C03625=1090.192,-119.581,450.543,174.558,16.064,152.527
C03626=1090.198,-119.332,450.534,174.560,16.065,152.526
C03627=1090.205,-119.082,450.524,174.562,16.066,152.526
C03628=1090.211,-118.832,450.515,174.563,16.066,152.526
C03629=1090.217,-118.582,450.505,174.565,16.066,152.526
C03630=1090.223,-118.332,450.496,174.567,16.067,152.525
C03631=1090.229,-118.082,450.487,174.568,16.067,152.525
C03632=1090.235,-117.832,450.477,174.570,16.068,152.525
C03633=1090.241,-117.583,450.468,174.571,16.069,152.525
C03634=1090.247,-117.333,450.458,174.573,16.069,152.525
C03635=1090.253,-117.084,450.449,174.574,16.070,152.524
C03636=1090.259,-116.834,450.439,174.576,16.070,152.524
C03637=1090.265,-116.584,450.430,174.577,16.070,152.524
C03638=1090.272,-116.334,450.420,174.579,16.071,152.524
C03639=1090.279,-116.085,450.411,174.580,16.071,152.523
C03640=1090.285,-115.835,450.402,174.582,16.072,152.523
C03641=1090.291,-115.585,450.392,174.584,16.073,152.523
C03642=1090.297,-115.335,450.382,174.585,16.073,152.523
C03643=1090.303,-115.086,450.373,174.587,16.073,152.522
C03644=1090.309,-114.836,450.364,174.589,16.074,152.522
C03645=1090.315,-114.587,450.354,174.590,16.074,152.522
C03646=1090.321,-114.337,450.345,174.592,16.075,152.522
C03647=1090.327,-114.087,450.335,174.594,16.076,152.522
C03648=1090.333,-113.837,450.325,174.595,16.076,152.521
C03649=1090.340,-113.587,450.316,174.597,16.076,152.521
C03650=1090.345,-113.318,450.306,174.598,16.077,152.521
C03651=1090.352,-113.049,450.295,174.600,16.078,152.521
C03652=1090.359,-112.781,450.285,174.601,16.078,152.521
C03653=1090.365,-112.512,450.275,174.603,16.079,152.520
C03654=1090.371,-112.262,450.265,174.605,16.080,152.520
C03655=1090.378,-112.012,450.256,174.607,16.080,152.520
C03656=1090.384,-111.762,450.246,174.608,16.080,152.519
C03657=1090.390,-111.513,450.236,174.610,16.081,152.519
C03658=1090.396,-111.263,450.226,174.612,16.082,152.519
C03659=1090.402,-111.013,450.216,174.613,16.082,152.519
C03660=1090.408,-110.763,450.207,174.615,16.083,152.519
C03661=1090.414,-110.514,450.197,174.616,16.084,152.519
C03662=1090.420,-110.264,450.188,174.617,16.084,152.518
C03663=1090.427,-110.014,450.178,174.619,16.085,152.518
C03664=1090.433,-109.764,450.168,174.621,16.085,152.518
C03665=1090.439,-109.514,450.159,174.622,16.086,152.518
C03666=1090.445,-109.265,450.149,174.624,16.086,152.517
C03667=1090.451,-109.015,450.140,174.626,16.087,152.517
C03668=1090.458,-108.766,450.130,174.627,16.087,152.517
C03669=1090.464,-108.516,450.120,174.628,16.088,152.517
C03670=1090.470,-108.266,450.110,174.630,16.089,152.517
C03671=1090.475,-108.016,450.100,174.632,16.089,152.516
C03672=1090.482,-107.766,450.091,174.633,16.089,152.516
C03673=1090.488,-107.516,450.081,174.635,16.091,152.516
C03674=1090.494,-107.266,450.072,174.637,16.091,152.516
C03675=1090.500,-107.017,450.061,174.638,16.091,152.515
C03676=1090.507,-106.767,450.052,174.640,16.092,152.515
C03677=1090.512,-106.517,450.041,174.641,16.093,152.515
C03678=1090.518,-106.268,450.032,174.643,16.093,152.515
C03679=1090.524,-106.018,450.023,174.644,16.094,152.515
C03680=1090.530,-105.769,450.013,174.646,16.095,152.515
C03681=1090.536,-105.519,450.003,174.648,16.096,152.514
C03682=1090.542,-105.269,449.993,174.649,16.096,152.514
C03683=1090.548,-105.020,449.983,174.651,16.097,152.514
C03684=1090.554,-104.770,449.974,174.653,16.097,152.514
C03685=1090.561,-104.521,449.963,174.653,16.098,152.514
C03686=1090.566,-104.271,449.953,174.655,16.099,152.513
C03687=1090.572,-104.021,449.944,174.657,16.099,152.513
C03688=1090.579,-103.771,449.934,174.659,16.100,152.513
C03689=1090.585,-103.521,449.924,174.660,16.100,152.513
C03690=1090.591,-103.272,449.914,174.662,16.101,152.512
C03691=1090.597,-103.022,449.904,174.663,16.102,152.512
C03692=1090.603,-102.772,449.894,174.665,16.103,152.512
C03693=1090.609,-102.522,449.885,174.666,16.103,152.512
C03694=1090.615,-102.273,449.874,174.668,16.104,152.512
C03695=1090.621,-102.023,449.864,174.670,16.105,152.511
C03696=1090.627,-101.773,449.855,174.672,16.106,152.511
C03697=1090.634,-101.523,449.844,174.673,16.106,152.511
C03698=1090.640,-101.273,449.834,174.675,16.106,152.511
C03699=1090.646,-101.023,449.824,174.676,16.108,152.511
C03700=1090.652,-100.774,449.814,174.677,16.108,152.511
C03701=1090.658,-100.524,449.805,174.679,16.108,152.510
C03702=1090.664,-100.274,449.794,174.681,16.109,152.510
C03703=1090.670,-100.024,449.785,174.683,16.110,152.510
C03704=1090.676,-99.775,449.775,174.684,16.111,152.510
C03705=1090.682,-99.525,449.764,174.685,16.111,152.510
C03706=1090.688,-99.276,449.754,174.687,16.112,152.509
C03707=1090.695,-99.026,449.745,174.689,16.113,152.509
C03708=1090.700,-98.776,449.734,174.690,16.113,152.509
C03709=1090.706,-98.527,449.724,174.692,16.114,152.509
C03710=1090.713,-98.277,449.715,174.694,16.115,152.509
C03711=1090.719,-98.027,449.705,174.696,16.115,152.508
C03712=1090.725,-97.778,449.694,174.696,16.116,152.508
C03713=1090.731,-97.528,449.685,174.698,16.117,152.508
C03714=1090.738,-97.252,449.673,174.700,16.118,152.508
C03715=1090.744,-96.976,449.662,174.702,16.118,152.508
C03716=1090.750,-96.701,449.651,174.703,16.120,152.508
C03717=1090.756,-96.425,449.640,174.705,16.120,152.507
C03718=1090.764,-96.175,449.629,174.707,16.121,152.507
C03719=1090.770,-95.925,449.619,174.709,16.122,152.507
C03720=1090.775,-95.676,449.608,174.710,16.123,152.507
C03721=1090.782,-95.426,449.599,174.712,16.123,152.507
C03722=1090.787,-95.176,449.589,174.713,16.124,152.506
C03723=1090.793,-94.927,449.578,174.715,16.125,152.506
C03724=1090.799,-94.677,449.568,174.716,16.126,152.506
C03725=1090.805,-94.427,449.558,174.718,16.126,152.506
C03726=1090.811,-94.177,449.548,174.719,16.127,152.506
C03727=1090.817,-93.928,449.538,174.721,16.128,152.505
C03728=1090.823,-93.678,449.527,174.723,16.129,152.505
C03729=1090.829,-93.429,449.517,174.724,16.129,152.505
C03730=1090.835,-93.179,449.507,174.726,16.130,152.505
C03731=1090.841,-92.930,449.497,174.727,16.131,152.505
C03732=1090.847,-92.680,449.487,174.729,16.132,152.505
C03733=1090.854,-92.430,449.476,174.731,16.133,152.504
C03734=1090.859,-92.180,449.466,174.732,16.133,152.504
C03735=1090.865,-91.930,449.455,174.734,16.134,152.504
C03736=1090.871,-91.680,449.445,174.735,16.135,152.504
C03737=1090.877,-91.431,449.434,174.737,16.136,152.504
C03738=1090.883,-91.181,449.425,174.739,16.137,152.504
C03739=1090.889,-90.931,449.414,174.740,16.137,152.504
C03740=1090.895,-90.682,449.404,174.742,16.138,152.503
C03741=1090.901,-90.432,449.394,174.743,16.139,152.503
C03742=1090.907,-90.182,449.384,174.745,16.140,152.503
C03743=1090.913,-89.932,449.373,174.747,16.141,152.503
C03744=1090.920,-89.683,449.362,174.748,16.141,152.503
C03745=1090.925,-89.433,449.352,174.749,16.142,152.502
C03746=1090.931,-89.184,449.342,174.751,16.143,152.502
C03747=1090.937,-88.934,449.332,174.753,16.144,152.502
C03748=1090.943,-88.684,449.321,174.755,16.145,152.502
C03749=1090.950,-88.434,449.310,174.756,16.145,152.502
C03750=1090.955,-88.184,449.300,174.757,16.146,152.502
C03751=1090.962,-87.935,449.290,174.759,16.147,152.501
C03752=1090.967,-87.685,449.280,174.761,16.148,152.501
C03753=1090.974,-87.436,449.269,174.762,16.149,152.501
C03754=1090.979,-87.186,449.259,174.763,16.149,152.501
C03755=1090.985,-86.935,449.248,174.765,16.150,152.501
C03756=1090.992,-86.686,449.238,174.767,16.151,152.501
C03757=1090.998,-86.437,449.227,174.769,16.152,152.500
C03758=1091.004,-86.187,449.217,174.771,16.153,152.500
C03759=1091.009,-85.937,449.206,174.772,16.154,152.500
C03760=1091.016,-85.687,449.195,174.773,16.154,152.500
C03761=1091.022,-85.437,449.186,174.775,16.155,152.500
C03762=1091.028,-85.188,449.175,174.776,16.156,152.500
C03763=1091.034,-84.939,449.164,174.778,16.157,152.499
C03764=1091.040,-84.689,449.154,174.780,16.158,152.499
C03765=1091.046,-84.438,449.143,174.782,16.159,152.499
C03766=1091.052,-84.189,449.133,174.783,16.159,152.499
C03767=1091.058,-83.940,449.122,174.784,16.160,152.499
C03768=1091.064,-83.690,449.112,174.786,16.161,152.499
C03769=1091.070,-83.440,449.101,174.788,16.162,152.498
C03770=1091.076,-83.190,449.090,174.789,16.163,152.498
C03771=1091.083,-82.941,449.080,174.791,16.164,152.498
C03772=1091.088,-82.691,449.070,174.792,16.164,152.498
C03773=1091.094,-82.442,449.059,174.794,16.165,152.498
C03774=1091.101,-82.192,449.048,174.796,16.166,152.498
C03775=1091.107,-81.942,449.037,174.797,16.167,152.498
C03776=1091.113,-81.692,449.028,174.799,16.168,152.497
C03777=1091.119,-81.443,449.017,174.801,16.169,152.497
C03778=1091.126,-81.170,449.005,174.803,16.170,152.497
C03779=1091.132,-80.896,448.993,174.804,16.171,152.497
C03780=1091.139,-80.623,448.981,174.806,16.172,152.497
C03781=1091.146,-80.349,448.970,174.808,16.173,152.496
C03782=1091.152,-80.099,448.960,174.809,16.174,152.496
C03783=1091.157,-79.850,448.949,174.811,16.175,152.496
C03784=1091.164,-79.600,448.937,174.812,16.175,152.496
C03785=1091.170,-79.350,448.927,174.814,16.176,152.496
C03786=1091.176,-79.101,448.916,174.815,16.177,152.496
C03787=1091.181,-78.851,448.906,174.817,16.178,152.496
C03788=1091.188,-78.601,448.895,174.819,16.179,152.495
C03789=1091.193,-78.351,448.884,174.820,16.180,152.495
C03790=1091.200,-78.102,448.874,174.822,16.181,152.495
C03791=1091.206,-77.852,448.863,174.823,16.181,152.495
C03792=1091.212,-77.602,448.852,174.825,16.183,152.495
C03793=1091.218,-77.353,448.841,174.826,16.184,152.495
C03794=1091.223,-77.103,448.831,174.828,16.184,152.495
C03795=1091.229,-76.853,448.820,174.830,16.185,152.494
C03796=1091.236,-76.603,448.809,174.832,16.187,152.494
C03797=1091.242,-76.354,448.798,174.833,16.187,152.494
C03798=1091.247,-76.104,448.787,174.835,16.188,152.494
C03799=1091.253,-75.855,448.776,174.837,16.190,152.494
C03800=1091.260,-75.605,448.765,174.837,16.190,152.494
C03801=1091.265,-75.355,448.754,174.839,16.191,152.494
C03802=1091.271,-75.106,448.743,174.841,16.192,152.493
C03803=1091.278,-74.856,448.733,174.843,16.193,152.493
C03804=1091.284,-74.606,448.722,174.844,16.194,152.493
C03805=1091.290,-74.357,448.711,174.846,16.195,152.493
C03806=1091.296,-74.107,448.700,174.848,16.196,152.493
C03807=1091.302,-73.857,448.689,174.849,16.197,152.493
C03808=1091.307,-73.608,448.678,174.851,16.198,152.493
C03809=1091.313,-73.358,448.668,174.852,16.198,152.492
C03810=1091.319,-73.108,448.657,174.854,16.199,152.492
C03811=1091.325,-72.858,448.646,174.855,16.201,152.492
C03812=1091.331,-72.608,448.635,174.857,16.202,152.492
C03813=1091.336,-72.359,448.624,174.859,16.203,152.492
C03814=1091.342,-72.109,448.613,174.860,16.204,152.492
C03815=1091.348,-71.859,448.602,174.862,16.205,152.492
C03816=1091.354,-71.610,448.591,174.864,16.206,152.491
C03817=1091.360,-71.360,448.580,174.865,16.207,152.491
C03818=1091.366,-71.110,448.568,174.867,16.208,152.491
C03819=1091.372,-70.861,448.557,174.868,16.209,152.491
C03820=1091.377,-70.611,448.546,174.869,16.210,152.491
C03821=1091.383,-70.362,448.535,174.871,16.210,152.491
C03822=1091.389,-70.112,448.524,174.873,16.212,152.491
C03823=1091.395,-69.862,448.513,174.874,16.213,152.491
C03824=1091.401,-69.613,448.502,174.876,16.214,152.491
C03825=1091.407,-69.362,448.491,174.878,16.215,152.490
C03826=1091.413,-69.113,448.480,174.879,16.216,152.490
C03827=1091.419,-68.863,448.469,174.881,16.217,152.490
C03828=1091.425,-68.613,448.458,174.883,16.218,152.490
C03829=1091.431,-68.364,448.447,174.884,16.219,152.490
C03830=1091.437,-68.114,448.436,174.886,16.220,152.490
C03831=1091.442,-67.864,448.424,174.888,16.221,152.490
C03832=1091.448,-67.615,448.413,174.889,16.222,152.490
C03833=1091.454,-67.365,448.402,174.891,16.224,152.489
C03834=1091.460,-67.115,448.390,174.892,16.224,152.489
C03835=1091.466,-66.866,448.380,174.894,16.225,152.489
C03836=1091.472,-66.616,448.369,174.895,16.226,152.489
C03837=1091.478,-66.366,448.357,174.897,16.227,152.489
C03838=1091.484,-66.117,448.347,174.898,16.228,152.489
C03839=1091.490,-65.868,448.335,174.900,16.229,152.489
C03840=1091.495,-65.617,448.323,174.902,16.230,152.488
C03841=1091.501,-65.368,448.312,174.903,16.231,152.488
C03842=1091.508,-65.097,448.300,174.905,16.232,152.488
C03843=1091.514,-64.825,448.288,174.907,16.233,152.488
C03844=1091.521,-64.555,448.276,174.908,16.235,152.488
C03845=1091.528,-64.283,448.264,174.911,16.236,152.488
C03846=1091.533,-64.033,448.253,174.912,16.237,152.488
C03847=1091.539,-63.784,448.241,174.913,16.237,152.488
C03848=1091.545,-63.534,448.229,174.915,16.239,152.487
C03849=1091.551,-63.284,448.218,174.917,16.240,152.487
C03850=1091.557,-63.034,448.207,174.918,16.241,152.487
C03851=1091.563,-62.785,448.196,174.920,16.242,152.487
C03852=1091.569,-62.536,448.185,174.921,16.243,152.487
C03853=1091.575,-62.286,448.173,174.923,16.244,152.487
C03854=1091.580,-62.036,448.162,174.925,16.245,152.487
C03855=1091.587,-61.786,448.150,174.927,16.246,152.487
C03856=1091.593,-61.537,448.139,174.928,16.247,152.486
C03857=1091.598,-61.287,448.128,174.930,16.248,152.486
C03858=1091.605,-61.037,448.117,174.931,16.249,152.486
C03859=1091.610,-60.788,448.105,174.933,16.251,152.486
C03860=1091.616,-60.538,448.094,174.935,16.252,152.486
C03861=1091.622,-60.288,448.083,174.936,16.253,152.486
C03862=1091.629,-60.039,448.071,174.938,16.254,152.486
C03863=1091.634,-59.789,448.060,174.940,16.255,152.486
C03864=1091.641,-59.539,448.049,174.941,16.256,152.485
C03865=1091.646,-59.290,448.036,174.943,16.257,152.485
C03866=1091.652,-59.039,448.025,174.945,16.258,152.485
C03867=1091.658,-58.790,448.014,174.946,16.259,152.485
C03868=1091.665,-58.540,448.002,174.948,16.260,152.485
C03869=1091.670,-58.291,447.991,174.949,16.262,152.485
C03870=1091.677,-58.041,447.979,174.951,16.262,152.485
C03871=1091.682,-57.792,447.968,174.953,16.263,152.485
C03872=1091.688,-57.542,447.957,174.955,16.264,152.484
C03873=1091.695,-57.293,447.945,174.956,16.266,152.484
C03874=1091.700,-57.042,447.933,174.958,16.267,152.484
C03875=1091.706,-56.793,447.922,174.959,16.268,152.484
C03876=1091.713,-56.543,447.911,174.961,16.269,152.484
C03877=1091.718,-56.293,447.900,174.963,16.270,152.484
C03878=1091.724,-56.044,447.887,174.964,16.271,152.484
C03879=1091.730,-55.794,447.876,174.966,16.272,152.484
C03880=1091.737,-55.544,447.864,174.968,16.273,152.483
C03881=1091.742,-55.295,447.853,174.969,16.274,152.483
C03882=1091.748,-55.045,447.841,174.971,16.275,152.483
C03883=1091.754,-54.796,447.830,174.973,16.276,152.483
C03884=1091.761,-54.546,447.818,174.974,16.278,152.483
C03885=1091.766,-54.297,447.807,174.976,16.279,152.483
C03886=1091.772,-54.047,447.795,174.977,16.280,152.483
C03887=1091.778,-53.797,447.784,174.979,16.281,152.483
C03888=1091.785,-53.548,447.772,174.981,16.282,152.482
C03889=1091.791,-53.297,447.761,174.983,16.283,152.482
C03890=1091.796,-53.048,447.748,174.984,16.284,152.482
C03891=1091.803,-52.798,447.737,174.986,16.285,152.482
C03892=1091.809,-52.549,447.725,174.987,16.286,152.482
C03893=1091.814,-52.299,447.714,174.989,16.287,152.482
C03894=1091.820,-52.050,447.702,174.991,16.289,152.482
C03895=1091.827,-51.800,447.691,174.992,16.290,152.482
C03896=1091.833,-51.550,447.679,174.994,16.290,152.481
C03897=1091.839,-51.301,447.667,174.996,16.291,152.481
C03898=1091.845,-51.051,447.655,174.997,16.293,152.481
C03899=1091.851,-50.802,447.644,174.999,16.294,152.481
C03900=1091.857,-50.551,447.632,175.001,16.295,152.481
C03901=1091.863,-50.302,447.620,175.002,16.296,152.481
C03902=1091.868,-50.052,447.609,175.004,16.297,152.481
C03903=1091.875,-49.802,447.597,175.005,16.298,152.481
C03904=1091.880,-49.553,447.584,175.007,16.299,152.481
C03905=1091.887,-49.303,447.573,175.009,16.301,152.480
C03906=1091.893,-49.034,447.560,175.010,16.302,152.480
C03907=1091.899,-48.763,447.547,175.012,16.303,152.480
C03908=1091.905,-48.493,447.535,175.013,16.304,152.480
C03909=1091.911,-48.224,447.522,175.016,16.306,152.480
C03910=1091.918,-47.974,447.510,175.017,16.307,152.480
C03911=1091.923,-47.724,447.498,175.019,16.308,152.480
C03912=1091.930,-47.475,447.486,175.021,16.309,152.480
C03913=1091.935,-47.225,447.474,175.022,16.310,152.480
C03914=1091.941,-46.975,447.462,175.024,16.311,152.480
C03915=1091.947,-46.726,447.451,175.026,16.313,152.479
C03916=1091.953,-46.476,447.438,175.027,16.314,152.479
C03917=1091.959,-46.227,447.426,175.029,16.315,152.479
C03918=1091.964,-45.977,447.415,175.030,16.316,152.479
C03919=1091.971,-45.727,447.403,175.032,16.317,152.479
C03920=1091.976,-45.478,447.391,175.034,16.318,152.479
C03921=1091.982,-45.228,447.379,175.035,16.319,152.479
C03922=1091.988,-44.978,447.367,175.037,16.320,152.479
C03923=1091.994,-44.729,447.355,175.038,16.322,152.479
C03924=1092.000,-44.479,447.343,175.040,16.323,152.478
C03925=1092.005,-44.229,447.331,175.042,16.324,152.478
C03926=1092.011,-43.979,447.319,175.043,16.325,152.478
C03927=1092.018,-43.730,447.307,175.045,16.326,152.478
C03928=1092.023,-43.481,447.295,175.046,16.327,152.478
C03929=1092.030,-43.231,447.283,175.048,16.328,152.478
C03930=1092.036,-42.981,447.271,175.050,16.330,152.478
C03931=1092.041,-42.731,447.259,175.052,16.331,152.478
C03932=1092.047,-42.482,447.247,175.054,16.332,152.478
C03933=1092.053,-42.231,447.235,175.055,16.334,152.477
C03934=1092.059,-41.983,447.223,175.057,16.335,152.477
C03935=1092.065,-41.733,447.211,175.059,16.336,152.477
C03936=1092.070,-41.483,447.198,175.060,16.337,152.477
C03937=1092.077,-41.234,447.187,175.062,16.338,152.477
C03938=1092.083,-40.984,447.174,175.063,16.339,152.477
C03939=1092.088,-40.734,447.162,175.065,16.340,152.477
C03940=1092.095,-40.485,447.151,175.067,16.342,152.477
C03941=1092.100,-40.235,447.138,175.068,16.343,152.477
C03942=1092.107,-39.985,447.126,175.070,16.344,152.477
C03943=1092.112,-39.736,447.114,175.071,16.345,152.476
C03944=1092.118,-39.486,447.101,175.073,16.346,152.476
C03945=1092.125,-39.237,447.089,175.075,16.347,152.476
C03946=1092.130,-38.987,447.077,175.077,16.349,152.476
C03947=1092.136,-38.737,447.065,175.079,16.350,152.476
C03948=1092.143,-38.487,447.053,175.080,16.351,152.476
C03949=1092.148,-38.238,447.041,175.082,16.352,152.476
C03950=1092.154,-37.988,447.029,175.084,16.354,152.476
C03951=1092.160,-37.738,447.016,175.085,16.355,152.476
C03952=1092.165,-37.489,447.004,175.087,16.356,152.476
C03953=1092.171,-37.239,446.991,175.088,16.357,152.475
C03954=1092.178,-36.990,446.979,175.090,16.358,152.475
C03955=1092.183,-36.741,446.967,175.092,16.359,152.475
C03956=1092.189,-36.491,446.955,175.093,16.360,152.475
C03957=1092.195,-36.241,446.942,175.095,16.362,152.475
C03958=1092.200,-35.992,446.930,175.097,16.364,152.475
C03959=1092.207,-35.742,446.918,175.099,16.365,152.475
C03960=1092.212,-35.492,446.905,175.100,16.366,152.475
C03961=1092.218,-35.243,446.893,175.102,16.367,152.475
C03962=1092.224,-34.993,446.881,175.103,16.368,152.475
C03963=1092.230,-34.743,446.868,175.105,16.369,152.474
C03964=1092.236,-34.493,446.855,175.107,16.371,152.474
C03965=1092.242,-34.244,446.844,175.108,16.372,152.474
C03966=1092.247,-33.995,446.831,175.110,16.373,152.474
C03967=1092.253,-33.745,446.819,175.111,16.374,152.474
C03968=1092.259,-33.495,446.807,175.114,16.376,152.474
C03969=1092.265,-33.246,446.794,175.115,16.377,152.474
C03970=1092.271,-32.976,446.781,175.117,16.378,152.474
C03971=1092.277,-32.707,446.767,175.119,16.379,152.474
C03972=1092.284,-32.437,446.754,175.120,16.380,152.474
C03973=1092.290,-32.167,446.740,175.123,16.382,152.473
C03974=1092.296,-31.918,446.728,175.124,16.383,152.473
C03975=1092.302,-31.668,446.715,175.126,16.385,152.473
C03976=1092.308,-31.418,446.703,175.127,16.386,152.473
C03977=1092.314,-31.168,446.690,175.129,16.387,152.473
C03978=1092.319,-30.919,446.678,175.130,16.388,152.473
C03979=1092.325,-30.669,446.666,175.132,16.389,152.473
C03980=1092.331,-30.420,446.653,175.135,16.391,152.473
C03981=1092.337,-30.170,446.641,175.136,16.392,152.473
C03982=1092.343,-29.920,446.627,175.138,16.393,152.473
C03983=1092.349,-29.671,446.615,175.139,16.394,152.472
C03984=1092.355,-29.422,446.603,175.141,16.396,152.472
C03985=1092.361,-29.172,446.591,175.143,16.397,152.472
C03986=1092.367,-28.922,446.578,175.144,16.398,152.472
C03987=1092.373,-28.672,446.565,175.146,16.399,152.472
C03988=1092.379,-28.423,446.553,175.147,16.400,152.472
C03989=1092.384,-28.174,446.540,175.150,16.402,152.472
C03990=1092.390,-27.924,446.527,175.151,16.403,152.472
C03991=1092.396,-27.674,446.515,175.153,16.404,152.472
C03992=1092.402,-27.424,446.502,175.155,16.405,152.472
C03993=1092.408,-27.175,446.489,175.156,16.406,152.471
C03994=1092.414,-26.925,446.477,175.158,16.408,152.471
C03995=1092.420,-26.676,446.464,175.160,16.409,152.471
C03996=1092.425,-26.426,446.452,175.161,16.410,152.471
C03997=1092.432,-26.176,446.439,175.163,16.412,152.471
C03998=1092.438,-25.927,446.426,175.165,16.413,152.471
C03999=1092.443,-25.677,446.414,175.166,16.414,152.471
C04000=1092.449,-25.427,446.401,175.168,16.416,152.471
C04001=1092.455,-25.178,446.388,175.170,16.417,152.471
C04002=1092.461,-24.928,446.375,175.171,16.418,152.471
C04003=1092.466,-24.678,446.362,175.173,16.419,152.471
C04004=1092.471,-24.429,446.350,175.175,16.421,152.470
C04005=1092.478,-24.180,446.337,175.177,16.422,152.470
C04006=1092.484,-23.930,446.324,175.179,16.423,152.470
C04007=1092.489,-23.680,446.312,175.180,16.424,152.470
C04008=1092.496,-23.431,446.298,175.181,16.426,152.470
C04009=1092.501,-23.181,446.286,175.183,16.427,152.470
C04010=1092.507,-22.932,446.274,175.185,16.428,152.470
C04011=1092.512,-22.682,446.260,175.187,16.430,152.470
C04012=1092.518,-22.432,446.247,175.189,16.431,152.470
C04013=1092.524,-22.182,446.235,175.190,16.432,152.470
C04014=1092.530,-21.933,446.221,175.192,16.433,152.469
C04015=1092.536,-21.683,446.209,175.194,16.434,152.469
C04016=1092.542,-21.435,446.196,175.195,16.435,152.469
C04017=1092.548,-21.185,446.183,175.198,16.437,152.469
C04018=1092.553,-20.934,446.170,175.199,16.438,152.469
C04019=1092.559,-20.685,446.157,175.201,16.439,152.469
C04020=1092.565,-20.435,446.144,175.202,16.441,152.469
C04021=1092.571,-20.186,446.131,175.204,16.442,152.469
C04022=1092.577,-19.936,446.119,175.205,16.443,152.469
C04023=1092.583,-19.686,446.106,175.208,16.445,152.469
C04024=1092.589,-19.437,446.092,175.209,16.446,152.469
C04025=1092.595,-19.187,446.080,175.211,16.447,152.468
C04026=1092.600,-18.938,446.067,175.213,16.448,152.468
C04027=1092.606,-18.688,446.054,175.214,16.450,152.468
C04028=1092.612,-18.439,446.041,175.216,16.451,152.468
C04029=1092.617,-18.189,446.028,175.217,16.452,152.468
C04030=1092.624,-17.940,446.014,175.220,16.454,152.468
C04031=1092.630,-17.690,446.002,175.221,16.455,152.468
C04032=1092.636,-17.440,445.989,175.223,16.456,152.468
C04033=1092.642,-17.191,445.976,175.225,16.457,152.468
C04034=1092.648,-16.921,445.962,175.227,16.459,152.467
C04035=1092.654,-16.650,445.947,175.229,16.460,152.467
C04036=1092.660,-16.379,445.934,175.230,16.461,152.467
C04037=1092.667,-16.109,445.919,175.233,16.463,152.467
C04038=1092.673,-15.859,445.906,175.234,16.464,152.467
C04039=1092.679,-15.610,445.893,175.236,16.465,152.467
C04040=1092.685,-15.361,445.880,175.237,16.467,152.467
C04041=1092.690,-15.110,445.867,175.239,16.468,152.467
C04042=1092.697,-14.861,445.853,175.241,16.469,152.467
C04043=1092.702,-14.612,445.841,175.243,16.471,152.467
C04044=1092.707,-14.362,445.827,175.245,16.472,152.466
C04045=1092.713,-14.112,445.815,175.246,16.473,152.466
C04046=1092.719,-13.863,445.801,175.248,16.474,152.466
C04047=1092.725,-13.614,445.788,175.249,16.475,152.466
C04048=1092.731,-13.364,445.775,175.252,16.477,152.466
C04049=1092.736,-13.114,445.761,175.253,16.478,152.466
C04050=1092.742,-12.864,445.749,175.255,16.479,152.466
C04051=1092.748,-12.615,445.735,175.256,16.481,152.466
C04052=1092.754,-12.365,445.721,175.258,16.482,152.466
C04053=1092.760,-12.115,445.709,175.260,16.484,152.466
C04054=1092.765,-11.866,445.695,175.262,16.485,152.466
C04055=1092.772,-11.617,445.682,175.264,16.486,152.465
C04056=1092.777,-11.366,445.669,175.265,16.487,152.465
C04057=1092.783,-11.117,445.655,175.267,16.488,152.465
C04058=1092.789,-10.868,445.642,175.269,16.490,152.465
C04059=1092.794,-10.618,445.629,175.271,16.491,152.465
C04060=1092.801,-10.368,445.616,175.272,16.492,152.465
C04061=1092.806,-10.119,445.602,175.274,16.493,152.465
C04062=1092.812,-9.870,445.589,175.276,16.494,152.465
C04063=1092.817,-9.619,445.575,175.278,16.496,152.465
C04064=1092.824,-9.370,445.562,175.279,16.498,152.465
C04065=1092.830,-9.121,445.549,175.281,16.499,152.465
C04066=1092.835,-8.871,445.536,175.283,16.500,152.464
C04067=1092.841,-8.621,445.522,175.284,16.501,152.464
C04068=1092.847,-8.372,445.509,175.287,16.503,152.464
C04069=1092.853,-8.123,445.495,175.288,16.504,152.464
C04070=1092.858,-7.873,445.481,175.290,16.505,152.464
C04071=1092.864,-7.623,445.469,175.292,16.506,152.464
C04072=1092.870,-7.374,445.455,175.293,16.508,152.464
C04073=1092.876,-7.124,445.442,175.296,16.509,152.464
C04074=1092.881,-6.875,445.428,175.297,16.510,152.464
C04075=1092.888,-6.625,445.415,175.299,16.512,152.463
C04076=1092.893,-6.375,445.401,175.300,16.513,152.463
C04077=1092.899,-6.126,445.388,175.302,16.514,152.463
C04078=1092.905,-5.876,445.374,175.304,16.516,152.463
C04079=1092.911,-5.626,445.361,175.306,16.517,152.463
C04080=1092.917,-5.377,445.347,175.308,16.518,152.463
C04081=1092.923,-5.128,445.334,175.309,16.519,152.463
C04082=1092.928,-4.877,445.320,175.312,16.521,152.463
C04083=1092.934,-4.628,445.307,175.313,16.522,152.463
C04084=1092.940,-4.379,445.293,175.315,16.523,152.462
C04085=1092.946,-4.129,445.280,175.317,16.524,152.462
C04086=1092.952,-3.880,445.266,175.318,16.525,152.462
C04087=1092.958,-3.631,445.253,175.321,16.527,152.462
C04088=1092.964,-3.380,445.239,175.322,16.528,152.462
C04089=1092.970,-3.131,445.225,175.324,16.529,152.462
C04090=1092.976,-2.881,445.212,175.325,16.530,152.462
C04091=1092.981,-2.632,445.198,175.328,16.533,152.462
C04092=1092.987,-2.382,445.184,175.329,16.534,152.462
C04093=1092.992,-2.132,445.171,175.331,16.535,152.462
C04094=1092.998,-1.883,445.157,175.332,16.536,152.462
C04095=1093.003,-1.633,445.143,175.335,16.538,152.461
C04096=1093.010,-1.384,445.130,175.336,16.539,152.461
C04097=1093.015,-1.134,445.116,175.338,16.540,152.461
C04098=1093.022,-0.862,445.101,175.340,16.541,152.461
C04099=1093.027,-0.590,445.086,175.342,16.543,152.461
C04100=1093.034,-0.318,445.071,175.344,16.544,152.461
C04101=1093.040,-0.047,445.056,175.346,16.546,152.461
C04102=1093.046,0.204,445.042,175.348,16.547,152.461
C04103=1093.052,0.453,445.029,175.349,16.548,152.461
C04104=1093.057,0.703,445.015,175.351,16.550,152.461
C04105=1093.063,0.952,445.001,175.353,16.551,152.460
C04106=1093.068,1.202,444.987,175.355,16.552,152.460
C04107=1093.075,1.451,444.974,175.356,16.554,152.460
C04108=1093.080,1.701,444.960,175.358,16.555,152.460
C04109=1093.086,1.950,444.946,175.360,16.556,152.460
C04110=1093.092,2.200,444.932,175.362,16.558,152.460
C04111=1093.097,2.449,444.917,175.364,16.559,152.460
C04112=1093.104,2.699,444.904,175.365,16.560,152.460
C04113=1093.109,2.948,444.890,175.368,16.562,152.460
C04114=1093.115,3.198,444.876,175.369,16.563,152.460
C04115=1093.120,3.447,444.863,175.371,16.564,152.459
C04116=1093.126,3.697,444.849,175.373,16.566,152.459
C04117=1093.132,3.947,444.835,175.375,16.567,152.459
C04118=1093.138,4.196,444.821,175.376,16.568,152.459
C04119=1093.143,4.446,444.807,175.378,16.569,152.459
C04120=1093.149,4.695,444.793,175.380,16.571,152.459
C04121=1093.155,4.945,444.779,175.382,16.572,152.459
C04122=1093.161,5.194,444.766,175.384,16.573,152.459
C04123=1093.167,5.444,444.751,175.385,16.574,152.459
C04124=1093.172,5.694,444.737,175.388,16.576,152.458
C04125=1093.178,5.943,444.724,175.389,16.577,152.458
C04126=1093.184,6.192,444.709,175.391,16.578,152.458
C04127=1093.189,6.442,444.695,175.393,16.579,152.458
C04128=1093.196,6.692,444.682,175.395,16.581,152.458
C04129=1093.201,6.941,444.668,175.397,16.582,152.458
C04130=1093.207,7.190,444.653,175.398,16.583,152.458
C04131=1093.213,7.440,444.639,175.400,16.584,152.458
C04132=1093.219,7.690,444.625,175.402,16.586,152.458
C04133=1093.224,7.940,444.611,175.404,16.587,152.457
C04134=1093.231,8.188,444.597,175.405,16.588,152.457
C04135=1093.236,8.438,444.583,175.407,16.590,152.457
C04136=1093.242,8.688,444.569,175.409,16.591,152.457
C04137=1093.248,8.938,444.555,175.411,16.592,152.457
C04138=1093.253,9.187,444.541,175.413,16.594,152.457
C04139=1093.259,9.436,444.527,175.415,16.595,152.457
C04140=1093.265,9.687,444.513,175.417,16.596,152.457
C04141=1093.271,9.935,444.498,175.418,16.597,152.457
C04142=1093.277,10.185,444.485,175.420,16.599,152.456
C04143=1093.283,10.435,444.470,175.422,16.600,152.456
C04144=1093.289,10.684,444.456,175.424,16.601,152.456
C04145=1093.294,10.934,444.442,175.426,16.602,152.456
C04146=1093.300,11.183,444.428,175.428,16.603,152.456
C04147=1093.306,11.433,444.413,175.430,16.605,152.456
C04148=1093.312,11.682,444.399,175.432,16.606,152.456
C04149=1093.317,11.932,444.385,175.433,16.607,152.456
C04150=1093.324,12.182,444.371,175.436,16.609,152.455
C04151=1093.329,12.431,444.357,175.437,16.610,152.455
C04152=1093.335,12.680,444.342,175.439,16.611,152.455
C04153=1093.341,12.930,444.328,175.440,16.612,152.455
C04154=1093.347,13.180,444.315,175.443,16.614,152.455
C04155=1093.353,13.429,444.300,175.444,16.615,152.455
C04156=1093.359,13.679,444.286,175.446,16.616,152.455
C04157=1093.365,13.928,444.271,175.449,16.618,152.455
C04158=1093.370,14.177,444.257,175.450,16.619,152.454
C04159=1093.377,14.427,444.242,175.452,16.620,152.454
C04160=1093.382,14.677,444.228,175.454,16.621,152.454
C04161=1093.388,14.926,444.214,175.456,16.623,152.454
C04162=1093.394,15.200,444.198,175.458,16.624,152.454
C04163=1093.400,15.474,444.183,175.460,16.626,152.454
C04164=1093.406,15.748,444.167,175.462,16.627,152.454
C04165=1093.413,16.022,444.151,175.464,16.628,152.454
C04166=1093.419,16.272,444.137,175.466,16.630,152.454
C04167=1093.424,16.521,444.122,175.467,16.631,152.453
C04168=1093.430,16.771,444.107,175.470,16.632,152.453
C04169=1093.436,17.020,444.093,175.471,16.634,152.453
C04170=1093.441,17.270,444.079,175.473,16.634,152.453
C04171=1093.448,17.520,444.064,175.476,16.636,152.453
C04172=1093.453,17.768,444.049,175.477,16.637,152.453
C04173=1093.459,18.018,444.036,175.479,16.638,152.453
C04174=1093.465,18.268,444.021,175.481,16.640,152.452
C04175=1093.470,18.518,444.006,175.483,16.641,152.452
C04176=1093.476,18.767,443.992,175.485,16.642,152.452
C04177=1093.482,19.017,443.977,175.487,16.644,152.452
C04178=1093.488,19.266,443.963,175.489,16.645,152.452
C04179=1093.494,19.515,443.948,175.490,16.646,152.452
C04180=1093.500,19.765,443.934,175.492,16.647,152.452
C04181=1093.505,20.014,443.919,175.495,16.649,152.452
C04182=1093.511,20.265,443.905,175.496,16.650,152.451
C04183=1093.516,20.514,443.890,175.498,16.651,152.451
C04184=1093.523,20.763,443.875,175.500,16.653,152.451
C04185=1093.528,21.013,443.861,175.502,16.654,152.451
C04186=1093.533,21.262,443.846,175.503,16.655,152.451
C04187=1093.540,21.512,443.831,175.506,16.657,152.451
C04188=1093.545,21.761,443.817,175.507,16.658,152.451
C04189=1093.551,22.010,443.803,175.509,16.658,152.451
C04190=1093.557,22.260,443.787,175.512,16.660,152.450
C04191=1093.562,22.509,443.772,175.513,16.661,152.450
C04192=1093.568,22.759,443.758,175.515,16.662,152.450
C04193=1093.574,23.009,443.743,175.517,16.664,152.450
C04194=1093.579,23.258,443.728,175.519,16.665,152.450
C04195=1093.585,23.508,443.714,175.521,16.666,152.450
C04196=1093.591,23.757,443.700,175.523,16.668,152.450
C04197=1093.597,24.007,443.684,175.525,16.669,152.450
C04198=1093.603,24.256,443.670,175.527,16.670,152.449
C04199=1093.609,24.506,443.655,175.529,16.672,152.449
C04200=1093.614,24.755,443.640,175.531,16.673,152.449
C04201=1093.620,25.005,443.625,175.532,16.674,152.449
C04202=1093.626,25.254,443.611,175.535,16.676,152.449
C04203=1093.632,25.503,443.596,175.537,16.676,152.449
C04204=1093.637,25.754,443.581,175.538,16.677,152.449
C04205=1093.643,26.002,443.567,175.541,16.679,152.448
C04206=1093.649,26.252,443.552,175.542,16.680,152.448
C04207=1093.654,26.501,443.537,175.544,16.681,152.448
C04208=1093.661,26.751,443.522,175.547,16.683,152.448
C04209=1093.666,27.000,443.507,175.548,16.684,152.448
C04210=1093.672,27.251,443.492,175.550,16.685,152.448
C04211=1093.677,27.500,443.478,175.552,16.687,152.448
C04212=1093.683,27.750,443.462,175.554,16.688,152.448
C04213=1093.689,27.998,443.447,175.556,16.688,152.447
C04214=1093.695,28.248,443.433,175.558,16.690,152.447
C04215=1093.700,28.497,443.417,175.560,16.691,152.447
C04216=1093.707,28.747,443.402,175.561,16.692,152.447
C04217=1093.713,28.996,443.388,175.564,16.694,152.447
C04218=1093.718,29.246,443.372,175.566,16.695,152.447
C04219=1093.724,29.496,443.358,175.567,16.696,152.447
C04220=1093.729,29.746,443.343,175.570,16.698,152.446
C04221=1093.735,29.994,443.328,175.571,16.699,152.446
C04222=1093.741,30.244,443.313,175.573,16.700,152.446
C04223=1093.746,30.493,443.298,175.575,16.702,152.446
C04224=1093.752,30.743,443.283,175.577,16.702,152.446
C04225=1093.758,30.992,443.268,175.579,16.703,152.446
C04226=1093.764,31.268,443.251,175.581,16.705,152.446
C04227=1093.770,31.543,443.234,175.584,16.707,152.445
C04228=1093.777,31.819,443.218,175.586,16.707,152.445
C04229=1093.783,32.094,443.201,175.588,16.709,152.445
C04230=1093.788,32.344,443.186,175.590,16.710,152.445
C04231=1093.795,32.593,443.171,175.592,16.712,152.445
C04232=1093.800,32.843,443.156,175.594,16.713,152.445
C04233=1093.806,33.092,443.141,175.596,16.714,152.444
C04234=1093.811,33.341,443.126,175.598,16.715,152.444
C04235=1093.817,33.591,443.111,175.600,16.717,152.444
C04236=1093.823,33.840,443.095,175.601,16.717,152.444
C04237=1093.829,34.089,443.080,175.604,16.719,152.444
C04238=1093.835,34.339,443.065,175.606,16.720,152.444
C04239=1093.840,34.589,443.049,175.607,16.721,152.444
C04240=1093.846,34.838,443.034,175.610,16.722,152.443
C04241=1093.851,35.088,443.019,175.611,16.724,152.443
C04242=1093.858,35.337,443.004,175.614,16.725,152.443
C04243=1093.863,35.587,442.989,175.616,16.726,152.443
C04244=1093.869,35.836,442.974,175.617,16.727,152.443
C04245=1093.875,36.086,442.958,175.620,16.729,152.443
C04246=1093.880,36.335,442.943,175.621,16.730,152.443
C04247=1093.886,36.584,442.928,175.623,16.731,152.442
C04248=1093.892,36.834,442.912,175.626,16.732,152.442
C04249=1093.898,37.083,442.898,175.627,16.733,152.442
C04250=1093.904,37.333,442.882,175.630,16.735,152.442
C04251=1093.910,37.582,442.867,175.632,16.736,152.442
C04252=1093.915,37.832,442.851,175.633,16.737,152.442
C04253=1093.921,38.082,442.836,175.636,16.738,152.441
C04254=1093.927,38.331,442.821,175.638,16.739,152.441
C04255=1093.932,38.581,442.806,175.639,16.740,152.441
C04256=1093.938,38.829,442.790,175.642,16.742,152.441
C04257=1093.943,39.079,442.774,175.644,16.743,152.441
C04258=1093.950,39.329,442.759,175.646,16.745,152.441
C04259=1093.955,39.578,442.744,175.648,16.745,152.440
C04260=1093.961,39.827,442.728,175.649,16.746,152.440
C04261=1093.966,40.077,442.712,175.652,16.748,152.440
C04262=1093.972,40.326,442.698,175.654,16.749,152.440
C04263=1093.978,40.576,442.682,175.656,16.750,152.440
C04264=1093.983,40.825,442.666,175.658,16.752,152.440
C04265=1093.989,41.075,442.651,175.659,16.753,152.440
C04266=1093.995,41.325,442.636,175.662,16.754,152.439
C04267=1094.001,41.573,442.620,175.664,16.755,152.439
C04268=1094.006,41.823,442.604,175.666,16.756,152.439
C04269=1094.012,42.073,442.589,175.668,16.757,152.439
C04270=1094.017,42.322,442.573,175.670,16.759,152.439
C04271=1094.024,42.571,442.558,175.672,16.760,152.438
C04272=1094.029,42.821,442.542,175.674,16.761,152.438
C04273=1094.035,43.070,442.527,175.676,16.762,152.438
C04274=1094.040,43.320,442.511,175.678,16.763,152.438
C04275=1094.047,43.570,442.496,175.680,16.764,152.438
C04276=1094.052,43.818,442.480,175.683,16.766,152.438
C04277=1094.058,44.068,442.465,175.684,16.767,152.438
C04278=1094.064,44.318,442.448,175.686,16.768,152.437
C04279=1094.069,44.567,442.433,175.689,16.769,152.437
C04280=1094.074,44.817,442.418,175.690,16.770,152.437
C04281=1094.080,45.066,442.401,175.693,16.772,152.437
C04282=1094.085,45.316,442.386,175.695,16.773,152.437
C04283=1094.091,45.565,442.370,175.697,16.774,152.437
C04284=1094.097,45.815,442.354,175.699,16.776,152.436
C04285=1094.102,46.063,442.339,175.700,16.776,152.436
C04286=1094.108,46.313,442.323,175.703,16.778,152.436
C04287=1094.114,46.563,442.307,175.705,16.779,152.436
C04288=1094.119,46.812,442.292,175.707,16.780,152.436
C04289=1094.125,47.061,442.275,175.709,16.781,152.436
C04290=1094.131,47.337,442.258,175.712,16.783,152.435
C04291=1094.137,47.612,442.241,175.713,16.784,152.435
C04292=1094.143,47.888,442.224,175.716,16.785,152.435
C04293=1094.150,48.164,442.206,175.718,16.787,152.435
C04294=1094.155,48.413,442.190,175.720,16.788,152.435
C04295=1094.161,48.662,442.174,175.723,16.789,152.434
C04296=1094.166,48.912,442.159,175.724,16.790,152.434
C04297=1094.172,49.162,442.142,175.726,16.791,152.434
C04298=1094.177,49.411,442.127,175.729,16.793,152.434
C04299=1094.183,49.660,442.111,175.730,16.793,152.434
C04300=1094.189,49.909,442.095,175.733,16.795,152.434
C04301=1094.194,50.159,442.080,175.734,16.796,152.433
C04302=1094.200,50.408,442.063,175.736,16.797,152.433
C04303=1094.206,50.658,442.048,175.739,16.798,152.433
C04304=1094.212,50.907,442.031,175.741,16.799,152.433
C04305=1094.218,51.157,442.015,175.743,16.801,152.433
C04306=1094.223,51.406,442.000,175.745,16.802,152.432
C04307=1094.229,51.655,441.984,175.747,16.803,152.432
C04308=1094.235,51.905,441.968,175.749,16.804,152.432
C04309=1094.240,52.155,441.952,175.751,16.805,152.432
C04310=1094.246,52.403,441.936,175.754,16.806,152.432
C04311=1094.252,52.653,441.920,175.755,16.807,152.432
C04312=1094.257,52.903,441.904,175.758,16.809,152.431
C04313=1094.263,53.152,441.887,175.760,16.810,152.431
C04314=1094.269,53.402,441.871,175.762,16.811,152.431
C04315=1094.274,53.650,441.855,175.764,16.812,152.431
C04316=1094.280,53.900,441.840,175.766,16.813,152.431
C04317=1094.285,54.150,441.824,175.769,16.814,152.430
C04318=1094.291,54.399,441.807,175.770,16.815,152.430
C04319=1094.297,54.649,441.792,175.773,16.816,152.430
C04320=1094.303,54.898,441.775,175.774,16.818,152.430
C04321=1094.308,55.147,441.760,175.777,16.819,152.430
C04322=1094.314,55.396,441.743,175.779,16.820,152.429
C04323=1094.320,55.646,441.726,175.782,16.821,152.429
C04324=1094.325,55.896,441.711,175.783,16.822,152.429
C04325=1094.331,56.145,441.695,175.785,16.823,152.429
C04326=1094.337,56.395,441.678,175.788,16.824,152.429
C04327=1094.343,56.644,441.662,175.789,16.825,152.428
C04328=1094.349,56.893,441.646,175.792,16.827,152.428
C04329=1094.354,57.142,441.630,175.794,16.827,152.428
C04330=1094.360,57.392,441.614,175.796,16.829,152.428
C04331=1094.365,57.642,441.598,175.798,16.830,152.428
C04332=1094.371,57.891,441.581,175.801,16.831,152.427
C04333=1094.377,58.140,441.565,175.803,16.832,152.427
C04334=1094.383,58.390,441.549,175.804,16.833,152.427
C04335=1094.389,58.639,441.533,175.807,16.834,152.427
C04336=1094.395,58.888,441.516,175.809,16.835,152.427
C04337=1094.400,59.138,441.499,175.812,16.836,152.426
C04338=1094.406,59.388,441.484,175.813,16.837,152.426
C04339=1094.412,59.637,441.468,175.816,16.839,152.426
C04340=1094.418,59.887,441.451,175.818,16.839,152.426
C04341=1094.423,60.135,441.436,175.820,16.840,152.425
C04342=1094.429,60.385,441.419,175.822,16.842,152.425
C04343=1094.434,60.634,441.402,175.824,16.842,152.425
C04344=1094.440,60.884,441.386,175.827,16.843,152.425
C04345=1094.446,61.133,441.370,175.829,16.844,152.425
C04346=1094.452,61.382,441.354,175.831,16.846,152.424
C04347=1094.458,61.632,441.337,175.833,16.846,152.424
C04348=1094.463,61.881,441.321,175.836,16.848,152.424
C04349=1094.469,62.131,441.304,175.837,16.849,152.424
C04350=1094.475,62.380,441.288,175.840,16.850,152.423
C04351=1094.481,62.629,441.272,175.842,16.851,152.423
C04352=1094.487,62.879,441.256,175.845,16.852,152.423
C04353=1094.492,63.128,441.239,175.846,16.853,152.423
C04354=1094.499,63.404,441.220,175.849,16.854,152.423
C04355=1094.505,63.679,441.202,175.851,16.855,152.422
C04356=1094.511,63.954,441.184,175.853,16.856,152.422
C04357=1094.518,64.230,441.166,175.856,16.857,152.422
C04358=1094.524,64.479,441.150,175.858,16.858,152.422
C04359=1094.530,64.728,441.133,175.861,16.859,152.421
C04360=1094.535,64.977,441.116,175.862,16.860,152.421
C04361=1094.541,65.227,441.099,175.865,16.862,152.421
C04362=1094.547,65.476,441.083,175.867,16.862,152.421
C04363=1094.553,65.726,441.066,175.870,16.864,152.420
C04364=1094.559,65.975,441.050,175.871,16.865,152.420
C04365=1094.564,66.225,441.033,175.874,16.866,152.420
C04366=1094.570,66.474,441.017,175.876,16.867,152.420
C04367=1094.575,66.723,440.999,175.879,16.868,152.419
C04368=1094.581,66.973,440.983,175.880,16.869,152.419
C04369=1094.587,67.222,440.967,175.883,16.870,152.419
C04370=1094.592,67.472,440.950,175.885,16.871,152.419
C04371=1094.598,67.721,440.934,175.887,16.872,152.419
C04372=1094.604,67.970,440.916,175.889,16.873,152.418
C04373=1094.610,68.219,440.900,175.891,16.874,152.418
C04374=1094.615,68.469,440.883,175.894,16.875,152.418
C04375=1094.621,68.718,440.867,175.896,16.876,152.418
C04376=1094.626,68.967,440.849,175.898,16.877,152.417
C04377=1094.632,69.217,440.833,175.900,16.878,152.417
C04378=1094.638,69.466,440.816,175.903,16.879,152.417
C04379=1094.644,69.716,440.800,175.905,16.880,152.417
C04380=1094.649,69.965,440.782,175.907,16.881,152.417
C04381=1094.655,70.214,440.766,175.909,16.882,152.416
C04382=1094.660,70.464,440.749,175.912,16.883,152.416
C04383=1094.666,70.713,440.733,175.914,16.884,152.416
C04384=1094.672,70.962,440.715,175.917,16.885,152.415
C04385=1094.678,71.211,440.699,175.918,16.886,152.415
C04386=1094.683,71.461,440.682,175.921,16.887,152.415
C04387=1094.688,71.710,440.665,175.923,16.888,152.415
C04388=1094.695,71.960,440.648,175.925,16.889,152.415
C04389=1094.700,72.210,440.631,175.927,16.890,152.414
C04390=1094.706,72.459,440.614,175.930,16.891,152.414
C04391=1094.712,72.708,440.597,175.932,16.892,152.414
C04392=1094.717,72.957,440.580,175.935,16.893,152.414
C04393=1094.723,73.207,440.564,175.936,16.894,152.413
C04394=1094.728,73.456,440.547,175.939,16.896,152.413
C04395=1094.734,73.705,440.529,175.941,16.896,152.413
C04396=1094.740,73.955,440.513,175.944,16.897,152.413
C04397=1094.745,74.204,440.495,175.945,16.898,152.412
C04398=1094.750,74.453,440.479,175.948,16.899,152.412
C04399=1094.757,74.703,440.461,175.950,16.900,152.412
C04400=1094.763,74.952,440.444,175.953,16.901,152.412
C04401=1094.768,75.202,440.428,175.955,16.902,152.411
C04402=1094.774,75.451,440.411,175.957,16.903,152.411
C04403=1094.779,75.701,440.394,175.959,16.904,152.411
C04404=1094.785,75.949,440.377,175.962,16.905,152.411
C04405=1094.791,76.199,440.360,175.964,16.906,152.410
C04406=1094.796,76.448,440.342,175.967,16.907,152.410
C04407=1094.802,76.698,440.325,175.969,16.908,152.410
C04408=1094.808,76.947,440.308,175.971,16.909,152.409
C04409=1094.814,77.197,440.291,175.973,16.909,152.409
C04410=1094.819,77.446,440.274,175.976,16.911,152.409
C04411=1094.825,77.694,440.257,175.978,16.911,152.409
C04412=1094.830,77.944,440.240,175.980,16.913,152.408
C04413=1094.837,78.194,440.222,175.982,16.913,152.408
C04414=1094.842,78.444,440.205,175.985,16.914,152.408
C04415=1094.848,78.692,440.188,175.987,16.915,152.408
C04416=1094.853,78.942,440.171,175.990,16.916,152.407
C04417=1094.859,79.191,440.154,175.992,16.917,152.407
C04418=1094.865,79.466,440.134,175.994,16.918,152.407
C04419=1094.871,79.741,440.116,175.997,16.919,152.407
C04420=1094.878,80.017,440.096,176.000,16.921,152.406
C04421=1094.884,80.291,440.078,176.002,16.922,152.406
C04422=1094.890,80.541,440.060,176.004,16.923,152.406
C04423=1094.895,80.790,440.043,176.007,16.924,152.406
C04424=1094.901,81.039,440.025,176.009,16.924,152.405
C04425=1094.906,81.289,440.008,176.012,16.926,152.405
C04426=1094.912,81.538,439.991,176.013,16.926,152.405
C04427=1094.918,81.788,439.973,176.016,16.928,152.404
C04428=1094.923,82.038,439.956,176.018,16.928,152.404
C04429=1094.928,82.287,439.938,176.021,16.930,152.404
C04430=1094.935,82.535,439.921,176.023,16.930,152.404
C04431=1094.940,82.785,439.905,176.025,16.931,152.403
C04432=1094.946,83.035,439.887,176.028,16.932,152.403
C04433=1094.952,83.284,439.869,176.030,16.933,152.403
C04434=1094.957,83.533,439.852,176.032,16.934,152.403
C04435=1094.962,83.782,439.835,176.035,16.935,152.402
C04436=1094.968,84.032,439.817,176.037,16.935,152.402
C04437=1094.974,84.281,439.799,176.039,16.937,152.402
C04438=1094.979,84.530,439.782,176.041,16.937,152.401
C04439=1094.985,84.779,439.764,176.044,16.939,152.401
C04440=1094.991,85.030,439.747,176.047,16.939,152.401
C04441=1094.996,85.279,439.729,176.049,16.940,152.401
C04442=1095.002,85.528,439.712,176.052,16.941,152.400
C04443=1095.007,85.777,439.694,176.054,16.942,152.400
C04444=1095.013,86.027,439.676,176.056,16.943,152.400
C04445=1095.019,86.276,439.659,176.058,16.944,152.399
C04446=1095.024,86.525,439.642,176.061,16.945,152.399
C04447=1095.030,86.774,439.625,176.063,16.945,152.399
C04448=1095.037,87.024,439.607,176.066,16.946,152.399
C04449=1095.042,87.273,439.589,176.068,16.947,152.398
C04450=1095.048,87.522,439.572,176.070,16.948,152.398
C04451=1095.054,87.772,439.554,176.073,16.948,152.398
C04452=1095.059,88.021,439.536,176.075,16.950,152.397
C04453=1095.065,88.270,439.519,176.078,16.951,152.397
C04454=1095.071,88.519,439.501,176.080,16.952,152.397
C04455=1095.076,88.768,439.483,176.083,16.952,152.396
C04456=1095.082,89.017,439.466,176.085,16.953,152.396
C04457=1095.088,89.267,439.448,176.087,16.954,152.396
C04458=1095.094,89.516,439.430,176.089,16.955,152.396
C04459=1095.099,89.765,439.413,176.092,16.956,152.395
C04460=1095.105,90.015,439.395,176.094,16.956,152.395
C04461=1095.110,90.264,439.376,176.097,16.958,152.395
C04462=1095.116,90.514,439.359,176.099,16.958,152.394
C04463=1095.122,90.763,439.341,176.102,16.959,152.394
C04464=1095.127,91.012,439.323,176.105,16.960,152.394
C04465=1095.133,91.262,439.305,176.106,16.961,152.393
C04466=1095.139,91.511,439.288,176.109,16.962,152.393
C04467=1095.144,91.760,439.270,176.111,16.962,152.393
C04468=1095.150,92.010,439.252,176.114,16.964,152.393
C04469=1095.155,92.259,439.234,176.116,16.964,152.392
C04470=1095.161,92.508,439.217,176.119,16.965,152.392
C04471=1095.167,92.758,439.199,176.121,16.966,152.392
C04472=1095.172,93.007,439.181,176.123,16.967,152.391
C04473=1095.178,93.256,439.164,176.126,16.968,152.391
C04474=1095.183,93.506,439.145,176.128,16.968,152.391
C04475=1095.189,93.754,439.127,176.131,16.970,152.390
C04476=1095.195,94.004,439.109,176.133,16.970,152.390
C04477=1095.201,94.253,439.091,176.136,16.971,152.390
C04478=1095.206,94.503,439.073,176.138,16.972,152.389
C04479=1095.212,94.752,439.055,176.141,16.972,152.389
C04480=1095.217,95.001,439.038,176.144,16.974,152.389
C04481=1095.223,95.251,439.020,176.145,16.974,152.389
C04482=1095.229,95.525,439.000,176.148,16.975,152.388
C04483=1095.235,95.801,438.980,176.151,16.976,152.388
C04484=1095.241,96.076,438.959,176.154,16.977,152.387
C04485=1095.247,96.352,438.940,176.156,16.978,152.387
C04486=1095.254,96.601,438.921,176.159,16.979,152.387
C04487=1095.259,96.850,438.904,176.162,16.980,152.386
C04488=1095.264,97.099,438.886,176.164,16.980,152.386
C04489=1095.270,97.349,438.868,176.167,16.981,152.386
C04490=1095.276,97.597,438.849,176.169,16.981,152.385
C04491=1095.282,97.847,438.831,176.171,16.983,152.385
C04492=1095.287,98.096,438.813,176.173,16.983,152.385
C04493=1095.293,98.346,438.795,176.176,16.984,152.384
C04494=1095.299,98.594,438.777,176.179,16.985,152.384
C04495=1095.304,98.845,438.758,176.181,16.986,152.384
C04496=1095.310,99.094,438.741,176.184,16.987,152.384
C04497=1095.316,99.343,438.722,176.186,16.987,152.383
C04498=1095.321,99.592,438.704,176.189,16.988,152.383
C04499=1095.327,99.842,438.686,176.192,16.989,152.382
C04500=1095.333,100.090,438.668,176.194,16.990,152.382
C04501=1095.338,100.340,438.649,176.197,16.990,152.382
C04502=1095.344,100.589,438.631,176.199,16.991,152.382
C04503=1095.350,100.838,438.613,176.202,16.992,152.381
C04504=1095.355,101.088,438.595,176.203,16.992,152.381
C04505=1095.362,101.337,438.576,176.206,16.993,152.380
C04506=1095.366,101.586,438.558,176.209,16.994,152.380
C04507=1095.373,101.835,438.540,176.211,16.995,152.380
C04508=1095.378,102.084,438.522,176.214,16.996,152.379
C04509=1095.384,102.334,438.503,176.216,16.996,152.379
C04510=1095.390,102.583,438.485,176.219,16.997,152.379
C04511=1095.395,102.833,438.467,176.222,16.998,152.378
C04512=1095.401,103.081,438.448,176.224,16.999,152.378
C04513=1095.406,103.331,438.430,176.227,17.000,152.378
C04514=1095.412,103.580,438.412,176.229,17.000,152.377
C04515=1095.417,103.830,438.393,176.232,17.001,152.377
C04516=1095.422,104.079,438.374,176.235,17.002,152.377
C04517=1095.429,104.328,438.356,176.237,17.002,152.376
C04518=1095.434,104.577,438.337,176.240,17.003,152.376
C04519=1095.440,104.827,438.319,176.241,17.004,152.376
C04520=1095.445,105.076,438.301,176.244,17.005,152.375
C04521=1095.451,105.325,438.282,176.247,17.005,152.375
C04522=1095.457,105.575,438.263,176.249,17.006,152.375
C04523=1095.462,105.823,438.245,176.252,17.007,152.374
C04524=1095.468,106.073,438.227,176.254,17.008,152.374
C04525=1095.474,106.322,438.208,176.257,17.008,152.374
C04526=1095.479,106.572,438.190,176.260,17.009,152.373
C04527=1095.484,106.820,438.171,176.262,17.010,152.373
C04528=1095.491,107.070,438.152,176.265,17.010,152.372
C04529=1095.496,107.320,438.134,176.267,17.011,152.372
C04530=1095.502,107.568,438.115,176.270,17.012,152.372
C04531=1095.507,107.817,438.096,176.273,17.013,152.371
C04532=1095.513,108.066,438.079,176.275,17.013,152.371
C04533=1095.519,108.316,438.059,176.278,17.014,152.371
C04534=1095.524,108.565,438.040,176.280,17.014,152.370
C04535=1095.530,108.814,438.023,176.283,17.015,152.370
C04536=1095.536,109.064,438.003,176.286,17.016,152.370
C04537=1095.542,109.313,437.985,176.288,17.017,152.369
C04538=1095.547,109.562,437.966,176.291,17.017,152.369
C04539=1095.552,109.812,437.947,176.293,17.017,152.368
C04540=1095.559,110.061,437.929,176.296,17.019,152.368
C04541=1095.564,110.310,437.910,176.299,17.020,152.368
C04542=1095.569,110.560,437.891,176.301,17.020,152.367
C04543=1095.576,110.809,437.873,176.304,17.020,152.367
C04544=1095.581,111.057,437.854,176.307,17.022,152.367
C04545=1095.587,111.307,437.835,176.309,17.022,152.366
C04546=1095.593,111.582,437.814,176.312,17.023,152.366
C04547=1095.599,111.857,437.793,176.315,17.023,152.365
C04548=1095.606,112.133,437.773,176.318,17.024,152.365
C04549=1095.612,112.408,437.752,176.321,17.025,152.364
C04550=1095.618,112.657,437.733,176.323,17.025,152.364
C04551=1095.623,112.906,437.714,176.326,17.026,152.364
C04552=1095.629,113.155,437.695,176.329,17.027,152.363
C04553=1095.634,113.405,437.677,176.331,17.027,152.363
C04554=1095.639,113.654,437.658,176.334,17.028,152.363
C04555=1095.645,113.903,437.638,176.336,17.028,152.362
C04556=1095.652,114.152,437.620,176.339,17.029,152.362
C04557=1095.657,114.402,437.601,176.342,17.030,152.361
C04558=1095.662,114.651,437.582,176.344,17.031,152.361
C04559=1095.668,114.900,437.562,176.347,17.031,152.361
C04560=1095.673,115.149,437.544,176.350,17.032,152.360
C04561=1095.679,115.398,437.524,176.352,17.032,152.360
C04562=1095.685,115.648,437.505,176.355,17.034,152.360
C04563=1095.690,115.897,437.486,176.358,17.034,152.359
C04564=1095.695,116.146,437.468,176.360,17.035,152.359
C04565=1095.701,116.396,437.448,176.363,17.035,152.358
C04566=1095.707,116.645,437.430,176.365,17.036,152.358
C04567=1095.712,116.894,437.411,176.368,17.037,152.358
C04568=1095.718,117.143,437.392,176.371,17.038,152.357
C04569=1095.724,117.393,437.372,176.373,17.038,152.357
C04570=1095.729,117.641,437.354,176.376,17.039,152.356
C04571=1095.734,117.891,437.334,176.379,17.039,152.356
C04572=1095.740,118.140,437.314,176.381,17.040,152.356
C04573=1095.746,118.389,437.295,176.384,17.040,152.355
C04574=1095.751,118.638,437.276,176.387,17.042,152.355
C04575=1095.757,118.887,437.257,176.389,17.042,152.355
C04576=1095.762,119.137,437.238,176.392,17.043,152.354
C04577=1095.768,119.386,437.218,176.395,17.043,152.354
C04578=1095.773,119.635,437.200,176.397,17.044,152.353
C04579=1095.779,119.884,437.180,176.400,17.044,152.353
C04580=1095.785,120.134,437.161,176.402,17.044,152.352
C04581=1095.790,120.383,437.142,176.405,17.045,152.352
C04582=1095.795,120.632,437.123,176.408,17.046,152.352
C04583=1095.801,120.881,437.103,176.410,17.046,152.351
C04584=1095.807,121.130,437.084,176.413,17.047,152.351
C04585=1095.813,121.379,437.065,176.416,17.048,152.350
C04586=1095.818,121.629,437.045,176.418,17.048,152.350
C04587=1095.824,121.878,437.026,176.421,17.049,152.350
C04588=1095.829,122.127,437.007,176.424,17.050,152.349
C04589=1095.835,122.376,436.987,176.427,17.050,152.349
C04590=1095.841,122.625,436.968,176.430,17.051,152.348
C04591=1095.847,122.875,436.949,176.433,17.051,152.348
C04592=1095.852,123.123,436.930,176.435,17.052,152.348
C04593=1095.858,123.372,436.910,176.438,17.052,152.347
C04594=1095.863,123.622,436.890,176.441,17.053,152.347
C04595=1095.868,123.871,436.871,176.443,17.053,152.346
C04596=1095.874,124.121,436.852,176.446,17.054,152.346
C04597=1095.880,124.370,436.832,176.449,17.055,152.345
C04598=1095.886,124.619,436.812,176.451,17.055,152.345
C04599=1095.891,124.868,436.794,176.454,17.056,152.345
C04600=1095.897,125.117,436.774,176.457,17.057,152.344
C04601=1095.902,125.366,436.754,176.459,17.056,152.344
C04602=1095.908,125.616,436.735,176.462,17.057,152.343
C04603=1095.914,125.864,436.715,176.465,17.058,152.343
C04604=1095.920,126.114,436.696,176.468,17.058,152.342
C04605=1095.926,126.363,436.677,176.471,17.059,152.342
C04606=1095.931,126.612,436.656,176.473,17.060,152.342
C04607=1095.936,126.862,436.637,176.476,17.060,152.341
C04608=1095.942,127.111,436.617,176.479,17.060,152.341
C04609=1095.948,127.359,436.598,176.482,17.061,152.340
C04610=1095.954,127.635,436.576,176.485,17.062,152.340
C04611=1095.961,127.911,436.555,176.487,17.061,152.339
C04612=1095.967,128.185,436.533,176.490,17.062,152.339
C04613=1095.973,128.461,436.511,176.494,17.063,152.338
C04614=1095.978,128.710,436.492,176.497,17.063,152.338
C04615=1095.984,128.959,436.472,176.500,17.064,152.337
C04616=1095.990,129.208,436.452,176.502,17.064,152.337
C04617=1095.996,129.457,436.432,176.505,17.065,152.337
C04618=1096.002,129.707,436.413,176.508,17.065,152.336
C04619=1096.007,129.956,436.393,176.510,17.066,152.336
C04620=1096.013,130.205,436.373,176.513,17.066,152.335
C04621=1096.019,130.454,436.353,176.516,17.067,152.335
C04622=1096.024,130.703,436.334,176.519,17.067,152.334
C04623=1096.030,130.952,436.314,176.522,17.068,152.334
C04624=1096.036,131.201,436.294,176.525,17.069,152.333
C04625=1096.041,131.451,436.274,176.527,17.068,152.333
C04626=1096.047,131.700,436.254,176.530,17.069,152.332
C04627=1096.053,131.949,436.235,176.533,17.070,152.332
C04628=1096.059,132.198,436.215,176.536,17.070,152.331
C04629=1096.064,132.447,436.195,176.538,17.070,152.331
C04630=1096.070,132.696,436.175,176.541,17.071,152.331
C04631=1096.076,132.945,436.155,176.545,17.071,152.330
C04632=1096.081,133.195,436.136,176.547,17.072,152.330
C04633=1096.087,133.444,436.116,176.550,17.072,152.329
C04634=1096.092,133.693,436.095,176.553,17.073,152.329
C04635=1096.098,133.942,436.076,176.555,17.073,152.328
C04636=1096.104,134.191,436.056,176.558,17.074,152.328
C04637=1096.109,134.440,436.035,176.561,17.075,152.327
C04638=1096.115,134.690,436.016,176.564,17.074,152.327
C04639=1096.120,134.939,435.996,176.567,17.075,152.327
C04640=1096.126,135.188,435.976,176.570,17.076,152.326
C04641=1096.132,135.436,435.956,176.573,17.076,152.326
C04642=1096.137,135.686,435.936,176.575,17.076,152.325
C04643=1096.143,135.935,435.916,176.578,17.077,152.325
C04644=1096.148,136.184,435.895,176.581,17.078,152.324
C04645=1096.154,136.433,435.875,176.583,17.078,152.324
C04646=1096.160,136.682,435.856,176.587,17.078,152.323
C04647=1096.165,136.932,435.836,176.590,17.079,152.323
C04648=1096.171,137.180,435.816,176.592,17.079,152.322
C04649=1096.176,137.429,435.795,176.595,17.079,152.322
C04650=1096.182,137.678,435.775,176.598,17.080,152.321
C04651=1096.187,137.928,435.755,176.601,17.080,152.321
C04652=1096.193,138.177,435.735,176.604,17.081,152.320
C04653=1096.199,138.426,435.715,176.607,17.081,152.320
C04654=1096.205,138.675,435.694,176.610,17.082,152.319
C04655=1096.210,138.925,435.674,176.612,17.082,152.319
C04656=1096.216,139.173,435.654,176.615,17.082,152.318
C04657=1096.222,139.423,435.633,176.618,17.083,152.318
C04658=1096.227,139.672,435.614,176.622,17.083,152.317
C04659=1096.233,139.921,435.594,176.624,17.084,152.317
C04660=1096.239,140.170,435.574,176.627,17.084,152.317
C04661=1096.244,140.419,435.553,176.630,17.085,152.316
C04662=1096.250,140.668,435.533,176.632,17.085,152.316
C04663=1096.256,140.918,435.512,176.635,17.085,152.315
C04664=1096.261,141.167,435.492,176.639,17.086,152.315
C04665=1096.267,141.416,435.472,176.642,17.086,152.314
C04666=1096.272,141.665,435.451,176.644,17.086,152.314
C04667=1096.278,141.914,435.431,176.647,17.087,152.313
C04668=1096.284,142.163,435.411,176.650,17.087,152.313
C04669=1096.289,142.412,435.390,176.652,17.088,152.312
C04670=1096.294,142.661,435.369,176.656,17.088,152.312
C04671=1096.301,142.910,435.349,176.659,17.089,152.311
C04672=1096.306,143.160,435.329,176.662,17.089,152.311
C04673=1096.311,143.409,435.308,176.664,17.089,152.310
C04674=1096.318,143.683,435.285,176.667,17.090,152.310
C04675=1096.324,143.958,435.263,176.671,17.090,152.309
C04676=1096.329,144.234,435.241,176.674,17.090,152.309
C04677=1096.336,144.509,435.218,176.677,17.090,152.308
C04678=1096.342,144.758,435.198,176.680,17.091,152.308
C04679=1096.347,145.007,435.177,176.683,17.092,152.307
C04680=1096.353,145.257,435.156,176.686,17.092,152.307
C04681=1096.359,145.505,435.136,176.689,17.092,152.306
C04682=1096.364,145.754,435.115,176.692,17.092,152.305
C04683=1096.370,146.003,435.094,176.695,17.093,152.305
C04684=1096.376,146.252,435.074,176.698,17.093,152.305
C04685=1096.382,146.502,435.053,176.701,17.094,152.304
C04686=1096.387,146.751,435.033,176.704,17.094,152.304
C04687=1096.392,147.000,435.012,176.707,17.094,152.303
C04688=1096.398,147.248,434.992,176.709,17.095,152.303
C04689=1096.404,147.498,434.971,176.712,17.095,152.302
C04690=1096.409,147.747,434.950,176.716,17.095,152.301
C04691=1096.415,147.996,434.930,176.719,17.096,152.301
C04692=1096.421,148.244,434.909,176.721,17.096,152.300
C04693=1096.427,148.494,434.888,176.724,17.096,152.300
C04694=1096.432,148.743,434.867,176.728,17.097,152.299
C04695=1096.437,148.992,434.847,176.731,17.097,152.299
C04696=1096.443,149.241,434.826,176.733,17.097,152.298
C04697=1096.449,149.491,434.805,176.736,17.097,152.298
C04698=1096.455,149.740,434.785,176.739,17.098,152.297
C04699=1096.460,149.988,434.764,176.743,17.099,152.297
C04700=1096.466,150.237,434.743,176.745,17.098,152.296
C04701=1096.471,150.487,434.722,176.748,17.099,152.296
C04702=1096.477,150.736,434.701,176.751,17.100,152.295
C04703=1096.482,150.985,434.680,176.755,17.100,152.295
C04704=1096.488,151.235,434.659,176.757,17.100,152.294
C04705=1096.494,151.483,434.638,176.760,17.100,152.294
C04706=1096.499,151.732,434.617,176.763,17.101,152.293
C04707=1096.504,151.981,434.597,176.767,17.101,152.293
C04708=1096.510,152.230,434.575,176.769,17.101,152.292
C04709=1096.516,152.480,434.555,176.772,17.102,152.292
C04710=1096.522,152.728,434.534,176.775,17.102,152.291
C04711=1096.528,152.978,434.513,176.778,17.102,152.291
C04712=1096.533,153.226,434.492,176.781,17.102,152.290
C04713=1096.539,153.475,434.471,176.784,17.102,152.289
C04714=1096.545,153.724,434.450,176.787,17.103,152.289
C04715=1096.550,153.974,434.429,176.790,17.104,152.288
C04716=1096.556,154.222,434.408,176.793,17.103,152.288
C04717=1096.561,154.472,434.387,176.796,17.104,152.287
C04718=1096.567,154.720,434.366,176.799,17.104,152.287
C04719=1096.572,154.970,434.345,176.803,17.104,152.286
C04720=1096.578,155.219,434.323,176.806,17.105,152.286
C04721=1096.584,155.468,434.303,176.808,17.105,152.285
C04722=1096.589,155.716,434.282,176.811,17.105,152.285
C04723=1096.595,155.966,434.261,176.815,17.106,152.284
C04724=1096.601,156.215,434.239,176.818,17.106,152.284
C04725=1096.606,156.464,434.219,176.820,17.106,152.283
C04726=1096.611,156.713,434.197,176.824,17.106,152.282
C04727=1096.617,156.962,434.175,176.827,17.107,152.282
C04728=1096.623,157.212,434.154,176.830,17.107,152.281
C04729=1096.628,157.460,434.133,176.832,17.107,152.281
C04730=1096.634,157.709,434.112,176.836,17.107,152.280
C04731=1096.640,157.959,434.091,176.839,17.108,152.280
C04732=1096.645,158.207,434.070,176.842,17.108,152.279
C04733=1096.651,158.457,434.049,176.845,17.108,152.279
C04734=1096.657,158.705,434.028,176.848,17.108,152.278
C04735=1096.662,158.954,434.006,176.851,17.108,152.278
C04736=1096.668,159.203,433.984,176.854,17.109,152.277
C04737=1096.673,159.452,433.964,176.858,17.109,152.276
C04738=1096.680,159.727,433.940,176.861,17.109,152.276
C04739=1096.686,160.002,433.916,176.864,17.110,152.275
C04740=1096.692,160.277,433.893,176.867,17.110,152.275
C04741=1096.698,160.552,433.869,176.871,17.110,152.274
C04742=1096.704,160.801,433.848,176.874,17.110,152.273
C04743=1096.709,161.050,433.826,176.877,17.111,152.273
C04744=1096.716,161.299,433.805,176.880,17.110,152.272
C04745=1096.721,161.548,433.783,176.883,17.111,152.272
C04746=1096.726,161.797,433.762,176.886,17.111,152.271
C04747=1096.732,162.046,433.741,176.890,17.111,152.271
C04748=1096.737,162.295,433.719,176.893,17.112,152.270
C04749=1096.743,162.544,433.697,176.895,17.112,152.270
C04750=1096.748,162.793,433.676,176.898,17.112,152.269
C04751=1096.753,163.042,433.654,176.901,17.113,152.269
C04752=1096.759,163.291,433.633,176.905,17.113,152.268
C04753=1096.765,163.540,433.612,176.908,17.113,152.267
C04754=1096.770,163.789,433.590,176.910,17.113,152.267
C04755=1096.776,164.038,433.568,176.914,17.114,152.266
C04756=1096.781,164.287,433.546,176.917,17.114,152.266
C04757=1096.787,164.536,433.525,176.920,17.114,152.265
C04758=1096.792,164.785,433.503,176.923,17.115,152.265
C04759=1096.798,165.034,433.481,176.926,17.114,152.264
C04760=1096.803,165.282,433.460,176.929,17.115,152.264
C04761=1096.809,165.532,433.438,176.932,17.115,152.263
C04762=1096.814,165.780,433.417,176.936,17.115,152.262
C04763=1096.820,166.030,433.394,176.939,17.116,152.262
C04764=1096.825,166.278,433.373,176.942,17.116,152.261
C04765=1096.830,166.528,433.351,176.945,17.116,152.261
C04766=1096.836,166.776,433.330,176.948,17.116,152.260
C04767=1096.841,167.026,433.307,176.951,17.117,152.260
C04768=1096.847,167.274,433.286,176.954,17.117,152.259
C04769=1096.852,167.524,433.264,176.958,17.117,152.258
C04770=1096.858,167.773,433.243,176.960,17.117,152.258
C04771=1096.863,168.022,433.220,176.963,17.117,152.257
C04772=1096.869,168.271,433.199,176.967,17.117,152.257
C04773=1096.874,168.520,433.177,176.970,17.118,152.256
C04774=1096.881,168.769,433.155,176.973,17.118,152.256
C04775=1096.885,169.018,433.133,176.977,17.118,152.255
C04776=1096.892,169.267,433.112,176.979,17.118,152.254
C04777=1096.897,169.515,433.089,176.982,17.119,152.254
C04778=1096.903,169.765,433.068,176.986,17.119,152.253
C04779=1096.908,170.013,433.046,176.989,17.119,152.253
C04780=1096.914,170.263,433.024,176.992,17.119,152.252
C04781=1096.919,170.512,433.002,176.996,17.120,152.251
C04782=1096.925,170.761,432.981,176.998,17.119,152.251
C04783=1096.931,171.010,432.958,177.001,17.120,152.250
C04784=1096.936,171.258,432.936,177.005,17.120,152.250
C04785=1096.942,171.508,432.914,177.008,17.120,152.249
C04786=1096.947,171.757,432.892,177.011,17.120,152.249
C04787=1096.953,172.006,432.871,177.015,17.121,152.248
C04788=1096.958,172.255,432.848,177.017,17.120,152.247
C04789=1096.964,172.503,432.826,177.020,17.121,152.247
C04790=1096.969,172.753,432.804,177.024,17.121,152.246
C04791=1096.976,173.001,432.782,177.027,17.121,152.246
C04792=1096.981,173.250,432.760,177.030,17.121,152.245
C04793=1096.986,173.499,432.738,177.034,17.121,152.244
C04794=1096.992,173.748,432.715,177.036,17.121,152.244
C04795=1096.997,173.997,432.693,177.040,17.121,152.243
C04796=1097.003,174.246,432.672,177.043,17.122,152.243
C04797=1097.009,174.495,432.649,177.046,17.122,152.242
C04798=1097.014,174.744,432.627,177.050,17.122,152.241
C04799=1097.020,174.993,432.605,177.053,17.122,152.241
C04800=1097.026,175.242,432.582,177.056,17.122,152.240
C04801=1097.031,175.491,432.560,177.059,17.122,152.240
C04802=1097.038,175.766,432.536,177.063,17.122,152.239
C04803=1097.044,176.040,432.512,177.067,17.123,152.238
C04804=1097.050,176.315,432.486,177.070,17.123,152.238
C04805=1097.056,176.589,432.463,177.074,17.123,152.237
C04806=1097.062,176.838,432.440,177.077,17.123,152.236
C04807=1097.068,177.086,432.418,177.080,17.122,152.236
C04808=1097.073,177.336,432.396,177.083,17.123,152.235
C04809=1097.079,177.585,432.373,177.086,17.123,152.234
C04810=1097.084,177.834,432.351,177.090,17.123,152.234
C04811=1097.090,178.082,432.329,177.093,17.123,152.233
C04812=1097.096,178.332,432.307,177.096,17.123,152.232
C04813=1097.101,178.581,432.284,177.100,17.124,152.232
C04814=1097.108,178.830,432.262,177.102,17.124,152.231
C04815=1097.113,179.079,432.239,177.106,17.123,152.231
C04816=1097.118,179.327,432.217,177.109,17.124,152.230
C04817=1097.125,179.576,432.195,177.112,17.124,152.229
C04818=1097.130,179.825,432.172,177.116,17.124,152.229
C04819=1097.136,180.074,432.150,177.119,17.124,152.228
C04820=1097.141,180.323,432.127,177.123,17.124,152.228
C04821=1097.147,180.571,432.105,177.125,17.124,152.227
C04822=1097.153,180.821,432.083,177.128,17.124,152.226
C04823=1097.158,181.070,432.060,177.132,17.124,152.226
C04824=1097.164,181.319,432.037,177.135,17.124,152.225
C04825=1097.170,181.568,432.015,177.139,17.124,152.224
C04826=1097.176,181.817,431.992,177.142,17.125,152.224
C04827=1097.182,182.066,431.969,177.146,17.125,152.223
C04828=1097.187,182.314,431.947,177.149,17.124,152.222
C04829=1097.193,182.563,431.925,177.152,17.124,152.222
C04830=1097.199,182.812,431.902,177.155,17.124,152.221
C04831=1097.205,183.061,431.879,177.158,17.125,152.221
C04832=1097.210,183.310,431.857,177.162,17.124,152.220
C04833=1097.216,183.559,431.834,177.165,17.125,152.219
C04834=1097.222,183.808,431.812,177.169,17.125,152.219
C04835=1097.228,184.057,431.789,177.172,17.125,152.218
C04836=1097.233,184.306,431.766,177.175,17.124,152.217
C04837=1097.239,184.554,431.744,177.178,17.124,152.217
C04838=1097.244,184.803,431.721,177.182,17.124,152.216
C04839=1097.251,185.052,431.699,177.185,17.125,152.215
C04840=1097.256,185.301,431.676,177.189,17.125,152.215
C04841=1097.261,185.550,431.652,177.192,17.125,152.214
C04842=1097.267,185.799,431.630,177.195,17.125,152.213
C04843=1097.273,186.048,431.607,177.199,17.125,152.213
C04844=1097.278,186.297,431.584,177.202,17.125,152.212
C04845=1097.283,186.545,431.561,177.205,17.125,152.212
C04846=1097.289,186.794,431.538,177.208,17.125,152.211
C04847=1097.295,187.043,431.515,177.211,17.125,152.210
C04848=1097.301,187.292,431.493,177.215,17.126,152.210
C04849=1097.306,187.541,431.470,177.218,17.126,152.209
C04850=1097.311,187.790,431.446,177.221,17.126,152.208
C04851=1097.316,188.038,431.423,177.225,17.126,152.208
C04852=1097.322,188.287,431.400,177.228,17.126,152.207
C04853=1097.328,188.537,431.378,177.232,17.126,152.206
C04854=1097.333,188.786,431.355,177.235,17.126,152.206
C04855=1097.339,189.035,431.332,177.238,17.126,152.205
C04856=1097.344,189.284,431.309,177.241,17.126,152.204
C04857=1097.350,189.533,431.286,177.244,17.126,152.204
C04858=1097.356,189.781,431.262,177.248,17.126,152.203
C04859=1097.362,190.030,431.239,177.251,17.127,152.203
C04860=1097.367,190.279,431.216,177.255,17.126,152.202
C04861=1097.372,190.527,431.194,177.258,17.126,152.201
C04862=1097.377,190.776,431.170,177.262,17.127,152.201
C04863=1097.383,191.025,431.147,177.265,17.127,152.200
C04864=1097.389,191.274,431.124,177.268,17.127,152.199
C04865=1097.395,191.523,431.101,177.272,17.127,152.199
C04866=1097.401,191.797,431.076,177.275,17.127,152.198
C04867=1097.407,192.072,431.050,177.279,17.127,152.197
C04868=1097.413,192.346,431.025,177.282,17.127,152.197
C04869=1097.419,192.619,430.999,177.286,17.127,152.196
C04870=1097.425,192.868,430.976,177.289,17.127,152.195
C04871=1097.430,193.118,430.952,177.293,17.127,152.195
C04872=1097.436,193.366,430.929,177.296,17.127,152.194
C04873=1097.442,193.615,430.906,177.300,17.127,152.193
C04874=1097.448,193.864,430.883,177.303,17.127,152.193
C04875=1097.453,194.113,430.859,177.307,17.127,152.192
C04876=1097.458,194.362,430.836,177.310,17.127,152.191
C04877=1097.464,194.611,430.813,177.313,17.128,152.191
C04878=1097.470,194.859,430.790,177.317,17.127,152.190
C04879=1097.475,195.108,430.766,177.320,17.127,152.189
C04880=1097.481,195.357,430.743,177.324,17.127,152.188
C04881=1097.487,195.606,430.720,177.327,17.128,152.188
C04882=1097.492,195.854,430.696,177.330,17.127,152.187
C04883=1097.498,196.103,430.673,177.333,17.127,152.187
C04884=1097.503,196.352,430.650,177.337,17.127,152.186
C04885=1097.509,196.601,430.626,177.340,17.127,152.185
C04886=1097.514,196.850,430.603,177.344,17.127,152.185
C04887=1097.521,197.099,430.579,177.347,17.127,152.184
C04888=1097.527,197.348,430.556,177.351,17.127,152.183
C04889=1097.532,197.597,430.532,177.354,17.127,152.182
C04890=1097.538,197.845,430.509,177.358,17.128,152.182
C04891=1097.543,198.094,430.485,177.361,17.127,152.181
C04892=1097.549,198.343,430.462,177.365,17.127,152.180
C04893=1097.555,198.592,430.438,177.368,17.127,152.180
C04894=1097.560,198.841,430.415,177.372,17.127,152.179
C04895=1097.566,199.090,430.391,177.375,17.127,152.178
C04896=1097.572,199.339,430.368,177.378,17.128,152.178
C04897=1097.577,199.587,430.344,177.382,17.128,152.177
C04898=1097.583,199.836,430.321,177.385,17.127,152.176
C04899=1097.589,200.084,430.297,177.388,17.127,152.176
C04900=1097.594,200.334,430.274,177.392,17.127,152.175
C04901=1097.600,200.582,430.250,177.395,17.127,152.174
C04902=1097.606,200.832,430.226,177.399,17.127,152.174
C04903=1097.612,201.080,430.202,177.402,17.127,152.173
C04904=1097.617,201.329,430.179,177.406,17.127,152.172
C04905=1097.623,201.578,430.155,177.409,17.127,152.172
C04906=1097.629,201.826,430.131,177.413,17.127,152.171
C04907=1097.634,202.076,430.108,177.416,17.127,152.170
C04908=1097.640,202.324,430.084,177.420,17.127,152.169
C04909=1097.645,202.573,430.060,177.423,17.127,152.169
C04910=1097.651,202.821,430.037,177.427,17.127,152.168
C04911=1097.657,203.070,430.012,177.430,17.127,152.167
C04912=1097.663,203.320,429.989,177.434,17.127,152.167
C04913=1097.668,203.568,429.965,177.437,17.127,152.166
C04914=1097.674,203.816,429.941,177.441,17.127,152.165
C04915=1097.679,204.066,429.918,177.444,17.127,152.165
C04916=1097.685,204.314,429.893,177.448,17.127,152.164
C04917=1097.691,204.563,429.869,177.451,17.127,152.163
C04918=1097.696,204.812,429.846,177.455,17.127,152.163
C04919=1097.702,205.061,429.822,177.458,17.127,152.162
C04920=1097.708,205.309,429.798,177.462,17.127,152.161
C04921=1097.713,205.558,429.774,177.465,17.127,152.161
C04922=1097.718,205.808,429.750,177.469,17.127,152.160
C04923=1097.725,206.056,429.726,177.472,17.127,152.159
C04924=1097.730,206.305,429.702,177.476,17.127,152.158
C04925=1097.735,206.553,429.678,177.479,17.127,152.158
C04926=1097.742,206.802,429.654,177.482,17.126,152.157
C04927=1097.747,207.051,429.630,177.485,17.126,152.156
C04928=1097.752,207.300,429.606,177.489,17.126,152.156
C04929=1097.758,207.548,429.582,177.492,17.126,152.155
C04930=1097.781,208.560,429.483,177.539,17.143,152.150
C04931=1097.790,208.931,429.448,177.544,17.145,152.149
C04932=1097.798,209.302,429.411,177.549,17.146,152.148
C04933=1097.806,209.673,429.374,177.553,17.147,152.148
C04934=1097.815,210.045,429.339,177.558,17.148,152.147
C04935=1097.820,210.293,429.314,177.562,17.149,152.146
C04936=1097.826,210.542,429.289,177.565,17.150,152.146
C04937=1097.832,210.791,429.265,177.568,17.151,152.145
C04938=1097.837,211.039,429.241,177.571,17.151,152.145
C04939=1097.843,211.288,429.216,177.575,17.153,152.145
C04940=1097.848,211.537,429.192,177.578,17.153,152.144
C04941=1097.854,211.786,429.167,177.581,17.154,152.144
C04942=1097.860,212.034,429.142,177.585,17.155,152.143
C04943=1097.865,212.283,429.118,177.588,17.156,152.143
C04944=1097.871,212.532,429.093,177.591,17.156,152.142
C04945=1097.876,212.781,429.069,177.594,17.157,152.142
C04946=1097.882,213.030,429.044,177.598,17.159,152.141
C04947=1097.888,213.278,429.020,177.601,17.159,152.141
C04948=1097.893,213.527,428.995,177.604,17.160,152.140
C04949=1097.899,213.776,428.971,177.608,17.161,152.140
C04950=1097.904,214.025,428.946,177.611,17.162,152.139
C04951=1097.910,214.273,428.921,177.614,17.163,152.139
C04952=1097.916,214.522,428.897,177.618,17.164,152.139
C04953=1097.921,214.771,428.872,177.621,17.165,152.138
C04954=1097.927,215.019,428.847,177.625,17.165,152.138
C04955=1097.932,215.268,428.823,177.628,17.167,152.137
C04956=1097.938,215.517,428.798,177.631,17.167,152.137
C04957=1097.943,215.765,428.773,177.634,17.168,152.136
C04958=1097.949,216.014,428.748,177.638,17.169,152.136
C04959=1097.955,216.262,428.723,177.641,17.170,152.135
C04960=1097.961,216.512,428.699,177.644,17.171,152.135
C04961=1097.966,216.760,428.674,177.647,17.172,152.134
C04962=1097.972,217.009,428.649,177.651,17.173,152.134
C04963=1097.977,217.258,428.625,177.654,17.173,152.134
C04964=1097.983,217.507,428.599,177.657,17.174,152.133
C04965=1097.988,217.755,428.575,177.661,17.175,152.133
C04966=1097.994,218.004,428.549,177.664,17.176,152.132
C04967=1098.000,218.252,428.525,177.668,17.177,152.132
C04968=1098.006,218.501,428.500,177.671,17.178,152.131
C04969=1098.010,218.750,428.475,177.674,17.179,152.131
C04970=1098.017,218.999,428.449,177.677,17.179,152.130
C04971=1098.022,219.247,428.425,177.681,17.181,152.130
C04972=1098.028,219.496,428.400,177.684,17.181,152.129
C04973=1098.034,219.745,428.375,177.687,17.182,152.129
C04974=1098.039,219.993,428.350,177.691,17.183,152.128
C04975=1098.045,220.243,428.325,177.694,17.184,152.128
C04976=1098.050,220.491,428.300,177.697,17.185,152.128
C04977=1098.057,220.739,428.275,177.701,17.186,152.127
C04978=1098.061,220.988,428.250,177.704,17.187,152.127
C04979=1098.067,221.237,428.224,177.708,17.187,152.126
C04980=1098.074,221.486,428.199,177.711,17.189,152.126
C04981=1098.079,221.734,428.175,177.715,17.189,152.125
C04982=1098.084,221.983,428.149,177.718,17.191,152.125
C04983=1098.093,222.358,428.112,177.723,17.192,152.124
C04984=1098.102,222.733,428.073,177.728,17.193,152.123
C04985=1098.110,223.109,428.035,177.733,17.195,152.123
C04986=1098.118,223.483,427.997,177.738,17.196,152.122
C04987=1098.124,223.732,427.973,177.741,17.197,152.122
C04988=1098.129,223.981,427.947,177.745,17.198,152.121
C04989=1098.135,224.230,427.921,177.748,17.199,152.121
C04990=1098.140,224.478,427.896,177.751,17.200,152.120
C04991=1098.146,224.727,427.870,177.755,17.201,152.120
C04992=1098.151,224.975,427.845,177.758,17.202,152.119
C04993=1098.157,225.224,427.820,177.761,17.203,152.119
C04994=1098.163,225.473,427.795,177.765,17.204,152.118
C04995=1098.168,225.721,427.769,177.768,17.205,152.118
C04996=1098.175,225.970,427.744,177.772,17.206,152.118
C04997=1098.180,226.219,427.718,177.775,17.207,152.117
C04998=1098.186,226.467,427.693,177.778,17.207,152.117
C04999=1098.191,226.716,427.668,177.782,17.208,152.116
C05000=1098.197,226.965,427.642,177.785,17.209,152.116
C05001=1098.202,227.214,427.617,177.788,17.210,152.115
C05002=1098.208,227.462,427.592,177.792,17.211,152.115
C05003=1098.213,227.711,427.566,177.795,17.212,152.114
C05004=1098.220,227.960,427.540,177.799,17.214,152.114
C05005=1098.225,228.208,427.515,177.802,17.214,152.114
C05006=1098.231,228.457,427.489,177.805,17.215,152.113
C05007=1098.236,228.706,427.463,177.809,17.216,152.113
C05008=1098.242,228.954,427.438,177.812,17.217,152.112
C05009=1098.247,229.202,427.413,177.816,17.218,152.112
C05010=1098.253,229.451,427.387,177.819,17.219,152.111
C05011=1098.259,229.700,427.361,177.822,17.220,152.111
C05012=1098.264,229.949,427.335,177.826,17.221,152.110
C05013=1098.270,230.196,427.310,177.829,17.222,152.110
C05014=1098.276,230.445,427.284,177.833,17.223,152.110
C05015=1098.282,230.694,427.258,177.835,17.224,152.109
C05016=1098.288,230.943,427.232,177.839,17.224,152.109
C05017=1098.292,231.191,427.207,177.842,17.226,152.108
C05018=1098.298,231.440,427.181,177.845,17.227,152.108
C05019=1098.304,231.689,427.156,177.849,17.228,152.107
C05020=1098.310,231.938,427.130,177.852,17.229,152.107
C05021=1098.315,232.186,427.103,177.855,17.230,152.106
C05022=1098.321,232.434,427.078,177.859,17.231,152.106
C05023=1098.326,232.683,427.052,177.862,17.232,152.106
C05024=1098.332,232.932,427.026,177.866,17.233,152.105
C05025=1098.338,233.181,427.000,177.869,17.234,152.105
C05026=1098.344,233.429,426.974,177.873,17.235,152.104
C05027=1098.349,233.678,426.949,177.876,17.236,152.104
C05028=1098.354,233.927,426.923,177.879,17.237,152.103
C05029=1098.360,234.175,426.896,177.883,17.238,152.103
C05030=1098.366,234.424,426.871,177.886,17.239,152.103
C05031=1098.372,234.673,426.845,177.890,17.240,152.102
C05032=1098.377,234.922,426.819,177.893,17.241,152.102
C05033=1098.382,235.169,426.793,177.896,17.243,152.101
C05034=1098.388,235.418,426.767,177.900,17.243,152.101
C05035=1098.396,235.785,426.728,177.904,17.245,152.100
C05036=1098.404,236.151,426.690,177.909,17.246,152.100
C05037=1098.413,236.518,426.652,177.914,17.248,152.099
C05038=1098.421,236.885,426.613,177.919,17.249,152.098
C05039=1098.427,237.133,426.586,177.923,17.251,152.098
C05040=1098.433,237.382,426.561,177.926,17.251,152.097
C05041=1098.438,237.629,426.535,177.930,17.253,152.097
C05042=1098.443,237.878,426.509,177.933,17.253,152.097
C05043=1098.449,238.127,426.482,177.937,17.255,152.096
C05044=1098.455,238.376,426.456,177.940,17.255,152.096
C05045=1098.460,238.624,426.429,177.944,17.257,152.095
C05046=1098.466,238.873,426.404,177.947,17.258,152.095
C05047=1098.472,239.121,426.377,177.950,17.259,152.094
C05048=1098.477,239.370,426.351,177.954,17.260,152.094
C05049=1098.483,239.619,426.324,177.957,17.261,152.094
C05050=1098.489,239.867,426.298,177.960,17.262,152.093
C05051=1098.494,240.116,426.272,177.963,17.263,152.093
C05052=1098.500,240.364,426.245,177.967,17.264,152.092
C05053=1098.505,240.613,426.219,177.970,17.265,152.092
C05054=1098.511,240.862,426.192,177.974,17.266,152.091
C05055=1098.517,241.110,426.166,177.977,17.267,152.091
C05056=1098.522,241.359,426.140,177.981,17.268,152.091
C05057=1098.528,241.607,426.113,177.984,17.269,152.090
C05058=1098.534,241.856,426.087,177.988,17.271,152.090
C05059=1098.539,242.105,426.061,177.991,17.272,152.089
C05060=1098.545,242.353,426.034,177.995,17.273,152.089
C05061=1098.551,242.601,426.007,177.998,17.274,152.088
C05062=1098.556,242.850,425.981,178.001,17.275,152.088
C05063=1098.562,243.099,425.955,178.004,17.276,152.088
C05064=1098.568,243.347,425.928,178.008,17.277,152.087
C05065=1098.574,243.596,425.901,178.011,17.278,152.087
C05066=1098.579,243.845,425.876,178.015,17.280,152.086
C05067=1098.585,244.093,425.849,178.018,17.280,152.086
C05068=1098.590,244.342,425.822,178.022,17.282,152.086
C05069=1098.596,244.590,425.795,178.025,17.283,152.085
C05070=1098.602,244.838,425.768,178.029,17.284,152.085
C05071=1098.607,245.087,425.742,178.032,17.285,152.084
C05072=1098.613,245.336,425.716,178.035,17.286,152.084
C05073=1098.618,245.584,425.689,178.038,17.287,152.083
C05074=1098.624,245.833,425.662,178.042,17.289,152.083
C05075=1098.629,246.081,425.635,178.045,17.290,152.083
C05076=1098.635,246.329,425.609,178.049,17.291,152.082
C05077=1098.641,246.578,425.582,178.052,17.292,152.082
C05078=1098.646,246.826,425.555,178.056,17.293,152.081
C05079=1098.652,247.075,425.528,178.059,17.294,152.081
C05080=1098.658,247.323,425.501,178.062,17.295,152.081
C05081=1098.663,247.571,425.475,178.065,17.296,152.080
C05082=1098.668,247.820,425.448,178.069,17.298,152.080
C05083=1098.674,248.069,425.421,178.072,17.299,152.079
C05084=1098.679,248.317,425.394,178.076,17.300,152.079
C05085=1098.685,248.566,425.367,178.079,17.301,152.079
C05086=1098.691,248.814,425.340,178.083,17.302,152.078
C05087=1098.699,249.175,425.301,178.088,17.304,152.078
C05088=1098.707,249.534,425.262,178.092,17.306,152.077
C05089=1098.715,249.894,425.223,178.097,17.308,152.077
C05090=1098.723,250.253,425.184,178.102,17.309,152.076
C05091=1098.729,250.501,425.157,178.105,17.311,152.076
C05092=1098.734,250.750,425.130,178.109,17.311,152.075
C05093=1098.739,250.998,425.103,178.112,17.313,152.075
C05094=1098.744,251.247,425.076,178.115,17.314,152.074
C05095=1098.751,251.496,425.049,178.119,17.315,152.074
C05096=1098.757,251.744,425.021,178.123,17.317,152.074
C05097=1098.762,251.993,424.994,178.126,17.318,152.073
C05098=1098.768,252.241,424.967,178.130,17.319,152.073
C05099=1098.773,252.490,424.940,178.132,17.320,152.072
C05100=1098.779,252.737,424.913,178.136,17.322,152.072
C05101=1098.784,252.986,424.886,178.139,17.322,152.072
C05102=1098.790,253.235,424.859,178.143,17.324,152.071
C05103=1098.795,253.484,424.831,178.146,17.325,152.071
C05104=1098.801,253.731,424.804,178.150,17.326,152.071
C05105=1098.806,253.980,424.777,178.153,17.328,152.070
C05106=1098.812,254.229,424.750,178.156,17.329,152.070
C05107=1098.818,254.477,424.722,178.160,17.330,152.069
C05108=1098.824,254.726,424.695,178.163,17.331,152.069
C05109=1098.829,254.974,424.668,178.167,17.333,152.069
C05110=1098.834,255.222,424.640,178.170,17.333,152.068
C05111=1098.841,255.471,424.613,178.174,17.335,152.068
C05112=1098.846,255.719,424.585,178.177,17.336,152.067
C05113=1098.852,255.968,424.558,178.180,17.337,152.067
C05114=1098.857,256.216,424.531,178.184,17.339,152.067
C05115=1098.863,256.465,424.503,178.187,17.340,152.066
C05116=1098.868,256.714,424.476,178.191,17.341,152.066
C05117=1098.875,256.961,424.449,178.194,17.342,152.065
C05118=1098.880,257.210,424.421,178.197,17.343,152.065
C05119=1098.886,257.459,424.393,178.201,17.345,152.065
C05120=1098.891,257.707,424.367,178.204,17.346,152.064
C05121=1098.897,257.955,424.339,178.208,17.347,152.064
C05122=1098.903,258.204,424.312,178.211,17.348,152.063
C05123=1098.908,258.452,424.284,178.215,17.350,152.063
C05124=1098.914,258.700,424.256,178.218,17.351,152.063
C05125=1098.920,258.949,424.229,178.221,17.352,152.062
C05126=1098.925,259.197,424.201,178.225,17.354,152.062
C05127=1098.930,259.446,424.173,178.228,17.355,152.062
C05128=1098.937,259.695,424.146,178.232,17.356,152.061
C05129=1098.942,259.943,424.118,178.235,17.357,152.061
C05130=1098.948,260.191,424.090,178.238,17.359,152.060
C05131=1098.954,260.440,424.063,178.242,17.360,152.060
C05132=1098.960,260.688,424.035,178.245,17.361,152.060
C05133=1098.965,260.936,424.008,178.249,17.362,152.059
C05134=1098.971,261.185,423.980,178.252,17.363,152.059
C05135=1098.977,261.433,423.952,178.256,17.365,152.058
C05136=1098.982,261.682,423.924,178.260,17.366,152.058
C05137=1098.988,261.930,423.897,178.262,17.367,152.058
C05138=1098.994,262.178,423.869,178.266,17.369,152.057
C05139=1099.002,262.535,423.829,178.271,17.370,152.057
C05140=1099.010,262.892,423.789,178.276,17.372,152.056
C05141=1099.019,263.249,423.749,178.281,17.374,152.056
C05142=1099.027,263.606,423.709,178.286,17.376,152.055
C05143=1099.033,263.854,423.681,178.289,17.377,152.055
C05144=1099.038,264.102,423.653,178.293,17.378,152.054
C05145=1099.045,264.350,423.625,178.296,17.379,152.054
C05146=1099.050,264.598,423.597,178.299,17.381,152.054
C05147=1099.056,264.848,423.570,178.303,17.383,152.053
C05148=1099.061,265.096,423.542,178.306,17.384,152.053
C05149=1099.067,265.345,423.513,178.310,17.385,152.053
C05150=1099.072,265.593,423.485,178.313,17.387,152.052
C05151=1099.078,265.841,423.458,178.316,17.388,152.052
C05152=1099.084,266.089,423.429,178.320,17.389,152.051
C05153=1099.089,266.337,423.401,178.323,17.390,152.051
C05154=1099.095,266.586,423.373,178.327,17.392,152.051
C05155=1099.100,266.834,423.345,178.330,17.393,152.050
C05156=1099.106,267.083,423.317,178.333,17.394,152.050
C05157=1099.112,267.331,423.289,178.337,17.396,152.050
C05158=1099.117,267.580,423.260,178.341,17.397,152.049
C05159=1099.123,267.828,423.232,178.344,17.398,152.049
C05160=1099.129,268.077,423.204,178.347,17.400,152.049
C05161=1099.134,268.325,423.176,178.351,17.402,152.048
C05162=1099.140,268.573,423.147,178.354,17.403,152.048
C05163=1099.146,268.821,423.119,178.358,17.404,152.048
C05164=1099.152,269.070,423.091,178.361,17.406,152.047
C05165=1099.157,269.318,423.063,178.364,17.407,152.047
C05166=1099.163,269.566,423.035,178.368,17.408,152.046
C05167=1099.168,269.814,423.007,178.371,17.410,152.046
C05168=1099.174,270.063,422.978,178.374,17.411,152.046
C05169=1099.180,270.311,422.950,178.378,17.413,152.045
C05170=1099.186,270.559,422.921,178.382,17.414,152.045
C05171=1099.191,270.807,422.893,178.385,17.415,152.045
C05172=1099.197,271.056,422.865,178.388,17.417,152.044
C05173=1099.202,271.304,422.836,178.392,17.419,152.044
C05174=1099.208,271.553,422.807,178.395,17.420,152.044
C05175=1099.213,271.801,422.779,178.399,17.421,152.043
C05176=1099.219,272.049,422.751,178.402,17.423,152.043
C05177=1099.225,272.297,422.722,178.405,17.424,152.043
C05178=1099.231,272.546,422.694,178.409,17.425,152.042
C05179=1099.236,272.795,422.665,178.413,17.427,152.042
C05180=1099.242,273.042,422.636,178.415,17.428,152.042
C05181=1099.248,273.291,422.608,178.419,17.430,152.041
C05182=1099.253,273.539,422.580,178.423,17.431,152.041
C05183=1099.259,273.787,422.551,178.426,17.432,152.041
C05184=1099.264,274.036,422.522,178.429,17.434,152.040
C05185=1099.270,274.284,422.494,178.433,17.436,152.040
C05186=1099.276,274.532,422.465,178.436,17.437,152.040
C05187=1099.282,274.780,422.437,178.439,17.439,152.040
C05188=1099.287,275.029,422.408,178.443,17.440,152.039
C05189=1099.293,275.278,422.379,178.447,17.442,152.039
C05190=1099.298,275.525,422.351,178.449,17.443,152.039
C05191=1099.306,275.884,422.308,178.455,17.445,152.038
C05192=1099.314,276.244,422.267,178.459,17.448,152.038
C05193=1099.323,276.604,422.226,178.464,17.449,152.037
C05194=1099.331,276.963,422.184,178.470,17.452,152.037
C05195=1099.336,277.212,422.155,178.473,17.453,152.036
C05196=1099.343,277.460,422.126,178.476,17.455,152.036
C05197=1099.348,277.707,422.097,178.480,17.456,152.036
C05198=1099.353,277.956,422.068,178.483,17.458,152.035
C05199=1099.360,278.205,422.039,178.486,17.459,152.035
C05200=1099.364,278.453,422.011,178.490,17.461,152.035
C05201=1099.370,278.701,421.982,178.493,17.463,152.034
C05202=1099.377,278.949,421.953,178.496,17.464,152.034
C05203=1099.382,279.197,421.924,178.500,17.465,152.034
C05204=1099.388,279.446,421.895,178.503,17.467,152.034
C05205=1099.393,279.694,421.866,178.507,17.469,152.033
C05206=1099.399,279.942,421.837,178.510,17.470,152.033
C05207=1099.404,280.191,421.808,178.514,17.472,152.033
C05208=1099.410,280.439,421.779,178.517,17.473,152.032
C05209=1099.416,280.687,421.749,178.521,17.475,152.032
C05210=1099.421,280.935,421.721,178.524,17.476,152.032
C05211=1099.428,281.183,421.692,178.527,17.478,152.031
C05212=1099.433,281.432,421.663,178.531,17.480,152.031
C05213=1099.438,281.680,421.633,178.534,17.482,152.031
C05214=1099.444,281.928,421.604,178.537,17.483,152.030
C05215=1099.449,282.176,421.575,178.541,17.484,152.030
C05216=1099.456,282.424,421.546,178.544,17.486,152.030
C05217=1099.461,282.673,421.516,178.548,17.488,152.030
C05218=1099.466,282.921,421.487,178.551,17.489,152.029
C05219=1099.472,283.169,421.458,178.554,17.491,152.029
C05220=1099.478,283.418,421.429,178.558,17.492,152.029
C05221=1099.484,283.666,421.400,178.561,17.494,152.028
C05222=1099.489,283.914,421.371,178.564,17.495,152.028
C05223=1099.494,284.162,421.341,178.568,17.497,152.028
C05224=1099.501,284.410,421.312,178.571,17.499,152.028
C05225=1099.506,284.659,421.282,178.575,17.501,152.027
C05226=1099.511,284.906,421.253,178.578,17.502,152.027
C05227=1099.517,285.154,421.224,178.581,17.504,152.027
C05228=1099.523,285.403,421.194,178.585,17.506,152.027
C05229=1099.528,285.651,421.165,178.589,17.507,152.026
C05230=1099.534,285.899,421.136,178.592,17.509,152.026
C05231=1099.539,286.147,421.106,178.595,17.510,152.026
C05232=1099.545,286.396,421.077,178.598,17.512,152.025
C05233=1099.551,286.643,421.047,178.602,17.514,152.025
C05234=1099.557,286.892,421.017,178.606,17.516,152.025
C05235=1099.562,287.140,420.988,178.609,17.518,152.025
C05236=1099.569,287.388,420.959,178.612,17.519,152.024
C05237=1099.574,287.637,420.929,178.616,17.520,152.024
C05238=1099.579,287.884,420.900,178.619,17.522,152.024
C05239=1099.585,288.133,420.870,178.623,17.524,152.023
C05240=1099.591,288.380,420.840,178.625,17.525,152.023
C05241=1099.597,288.629,420.811,178.629,17.527,152.023
C05242=1099.602,288.877,420.781,178.633,17.529,152.023
C05243=1099.611,289.246,420.737,178.638,17.532,152.022
C05244=1099.619,289.616,420.693,178.642,17.534,152.022
C05245=1099.628,289.983,420.649,178.648,17.537,152.021
C05246=1099.636,290.352,420.604,178.653,17.539,152.021
C05247=1099.641,290.601,420.575,178.656,17.541,152.021
C05248=1099.647,290.849,420.544,178.659,17.542,152.020
C05249=1099.653,291.097,420.515,178.663,17.544,152.020
C05250=1099.659,291.345,420.486,178.666,17.546,152.020
C05251=1099.665,291.593,420.455,178.670,17.548,152.020
C05252=1099.670,291.842,420.426,178.673,17.550,152.019
C05253=1099.676,292.090,420.396,178.676,17.551,152.019
C05254=1099.682,292.338,420.366,178.680,17.553,152.019
C05255=1099.687,292.586,420.336,178.683,17.555,152.019
C05256=1099.692,292.833,420.306,178.687,17.557,152.018
C05257=1099.698,293.082,420.277,178.690,17.559,152.018
C05258=1099.704,293.330,420.246,178.694,17.560,152.018
C05259=1099.709,293.578,420.217,178.696,17.562,152.018
C05260=1099.715,293.826,420.186,178.700,17.564,152.018
C05261=1099.721,294.074,420.157,178.704,17.565,152.017
C05262=1099.726,294.322,420.126,178.707,17.567,152.017
C05263=1099.732,294.571,420.097,178.710,17.569,152.017
C05264=1099.738,294.818,420.066,178.714,17.571,152.017
C05265=1099.743,295.067,420.037,178.717,17.573,152.016
C05266=1099.749,295.315,420.006,178.720,17.575,152.016
C05267=1099.755,295.563,419.976,178.724,17.576,152.016
C05268=1099.760,295.811,419.946,178.727,17.578,152.016
C05269=1099.766,296.059,419.916,178.731,17.580,152.015
C05270=1099.772,296.307,419.886,178.734,17.582,152.015
C05271=1099.777,296.555,419.856,178.738,17.584,152.015
C05272=1099.783,296.803,419.826,178.741,17.586,152.015
C05273=1099.789,297.051,419.795,178.744,17.587,152.015
C05274=1099.794,297.299,419.765,178.747,17.589,152.014
C05275=1099.800,297.547,419.735,178.751,17.591,152.014
C05276=1099.806,297.795,419.704,178.754,17.593,152.014
C05277=1099.811,298.043,419.674,178.758,17.595,152.014
C05278=1099.817,298.292,419.644,178.761,17.597,152.013
C05279=1099.823,298.540,419.614,178.765,17.599,152.013
C05280=1099.828,298.788,419.583,178.768,17.601,152.013
C05281=1099.834,299.036,419.552,178.771,17.603,152.013
C05282=1099.840,299.284,419.523,178.774,17.605,152.013
C05283=1099.845,299.532,419.492,178.777,17.607,152.013
C05284=1099.851,299.780,419.461,178.781,17.609,152.012
C05285=1099.856,300.028,419.431,178.784,17.611,152.012
C05286=1099.862,300.276,419.401,178.788,17.613,152.012
C05287=1099.867,300.524,419.370,178.791,17.615,152.012
C05288=1099.873,300.772,419.339,178.795,17.617,152.012
C05289=1099.879,301.020,419.309,178.798,17.619,152.011
C05290=1099.884,301.268,419.279,178.801,17.621,152.011
C05291=1099.890,301.516,419.248,178.805,17.623,152.011
C05292=1099.895,301.764,419.217,178.808,17.625,152.011
C05293=1099.900,302.012,419.187,178.811,17.626,152.011
C05294=1099.906,302.260,419.157,178.814,17.628,152.010
C05295=1099.915,302.643,419.109,178.819,17.631,152.010
C05296=1099.924,303.025,419.062,178.825,17.635,152.010
C05297=1099.932,303.408,419.015,178.830,17.638,152.010
C05298=1099.941,303.791,418.967,178.836,17.641,152.009
C05299=1099.947,304.039,418.936,178.839,17.643,152.009
C05300=1099.952,304.287,418.905,178.842,17.645,152.009
C05301=1099.958,304.535,418.875,178.846,17.648,152.009
C05302=1099.964,304.783,418.844,178.848,17.649,152.009
C05303=1099.969,305.031,418.813,178.852,17.651,152.009
C05304=1099.975,305.279,418.783,178.855,17.653,152.008
C05305=1099.980,305.527,418.751,178.858,17.655,152.008
C05306=1099.986,305.775,418.721,178.862,17.657,152.008
C05307=1099.992,306.023,418.690,178.865,17.659,152.008
C05308=1099.997,306.271,418.659,178.869,17.661,152.008
C05309=1100.003,306.519,418.628,178.872,17.663,152.007
C05310=1100.009,306.767,418.597,178.875,17.666,152.007
C05311=1100.014,307.015,418.566,178.879,17.668,152.007
C05312=1100.020,307.263,418.536,178.882,17.670,152.007
C05313=1100.025,307.511,418.505,178.885,17.672,152.007
C05314=1100.031,307.759,418.474,178.889,17.674,152.007
C05315=1100.036,308.007,418.443,178.892,17.676,152.007
C05316=1100.043,308.255,418.412,178.896,17.678,152.006
C05317=1100.048,308.503,418.380,178.899,17.680,152.006
C05318=1100.054,308.750,418.350,178.902,17.682,152.006
C05319=1100.060,308.999,418.319,178.906,17.684,152.006
C05320=1100.066,309.247,418.288,178.909,17.687,152.006
C05321=1100.071,309.495,418.257,178.912,17.689,152.006
C05322=1100.077,309.743,418.225,178.916,17.691,152.005
C05323=1100.083,309.991,418.194,178.919,17.693,152.005
C05324=1100.088,310.238,418.163,178.923,17.695,152.005
C05325=1100.094,310.486,418.132,178.926,17.697,152.005
C05326=1100.100,310.735,418.101,178.929,17.700,152.005
C05327=1100.105,310.982,418.069,178.933,17.702,152.005
C05328=1100.111,311.231,418.039,178.936,17.704,152.005
C05329=1100.117,311.478,418.007,178.939,17.706,152.004
C05330=1100.123,311.726,417.976,178.943,17.708,152.004
C05331=1100.129,311.974,417.944,178.946,17.710,152.004
C05332=1100.134,312.222,417.913,178.949,17.712,152.004
C05333=1100.140,312.470,417.882,178.953,17.714,152.004
C05334=1100.146,312.718,417.850,178.956,17.717,152.004
C05335=1100.151,312.966,417.820,178.959,17.719,152.004
C05336=1100.158,313.214,417.788,178.963,17.721,152.004
C05337=1100.163,313.462,417.756,178.966,17.723,152.003
C05338=1100.169,313.710,417.725,178.969,17.725,152.003
C05339=1100.175,313.958,417.694,178.973,17.727,152.003
C05340=1100.181,314.206,417.662,178.976,17.729,152.003
C05341=1100.186,314.454,417.631,178.979,17.732,152.003
C05342=1100.192,314.701,417.600,178.983,17.734,152.003
C05343=1100.198,314.949,417.568,178.986,17.736,152.003
C05344=1100.203,315.197,417.537,178.989,17.738,152.002
C05345=1100.209,315.446,417.505,178.993,17.741,152.002
C05346=1100.214,315.693,417.473,178.996,17.743,152.002
C05347=1100.224,316.079,417.424,179.001,17.746,152.002
C05348=1100.232,316.464,417.375,179.005,17.750,152.002
C05349=1100.241,316.850,417.326,179.011,17.754,152.002
C05350=1100.249,317.235,417.277,179.016,17.757,152.002
C05351=1100.255,317.483,417.245,179.019,17.760,152.002
C05352=1100.260,317.730,417.213,179.022,17.762,152.002
C05353=1100.266,317.978,417.181,179.026,17.765,152.002
C05354=1100.272,318.227,417.150,179.029,17.767,152.002
C05355=1100.277,318.474,417.118,179.032,17.769,152.001
C05356=1100.283,318.722,417.086,179.035,17.771,152.001
C05357=1100.288,318.970,417.055,179.039,17.774,152.001
C05358=1100.294,319.218,417.023,179.042,17.776,152.001
C05359=1100.300,319.466,416.991,179.045,17.779,152.001
C05360=1100.306,319.714,416.959,179.048,17.781,152.001
C05361=1100.311,319.961,416.927,179.052,17.784,152.001
C05362=1100.316,320.210,416.895,179.055,17.786,152.001
C05363=1100.322,320.457,416.863,179.059,17.788,152.001
C05364=1100.328,320.706,416.831,179.062,17.791,152.001
C05365=1100.333,320.953,416.799,179.065,17.793,152.001
C05366=1100.339,321.201,416.767,179.068,17.796,152.001
C05367=1100.344,321.449,416.736,179.071,17.798,152.001
C05368=1100.350,321.697,416.704,179.075,17.801,152.001
C05369=1100.356,321.945,416.672,179.078,17.803,152.001
C05370=1100.361,322.193,416.639,179.081,17.805,152.001
C05371=1100.367,322.441,416.607,179.084,17.808,152.001
C05372=1100.373,322.688,416.575,179.088,17.811,152.000
C05373=1100.379,322.937,416.543,179.091,17.813,152.000
C05374=1100.384,323.184,416.511,179.094,17.816,152.000
C05375=1100.390,323.432,416.479,179.098,17.818,152.000
C05376=1100.395,323.681,416.447,179.101,17.820,152.000
C05377=1100.401,323.928,416.414,179.104,17.823,152.000
C05378=1100.407,324.176,416.382,179.107,17.825,152.000
C05379=1100.412,324.423,416.351,179.110,17.828,152.000
C05380=1100.418,324.672,416.319,179.114,17.830,152.000
C05381=1100.424,324.920,416.285,179.117,17.833,152.000
C05382=1100.429,325.167,416.254,179.121,17.836,152.000
C05383=1100.435,325.415,416.222,179.124,17.838,152.000
C05384=1100.442,325.663,416.189,179.127,17.840,152.000
C05385=1100.447,325.910,416.157,179.130,17.843,152.000
C05386=1100.452,326.159,416.125,179.133,17.846,152.000
C05387=1100.458,326.406,416.092,179.136,17.848,152.000
C05388=1100.464,326.654,416.060,179.139,17.850,152.000
C05389=1100.469,326.902,416.028,179.143,17.853,152.000
C05390=1100.475,327.150,415.995,179.147,17.856,152.000
C05391=1100.481,327.398,415.963,179.150,17.858,152.000
C05392=1100.487,327.645,415.930,179.153,17.861,152.000
C05393=1100.492,327.894,415.898,179.156,17.864,152.000
C05394=1100.499,328.141,415.865,179.159,17.866,152.000
C05395=1100.505,328.390,415.833,179.162,17.868,152.000
C05396=1100.509,328.637,415.801,179.166,17.871,152.000
C05397=1100.516,328.885,415.768,179.169,17.874,152.000
C05398=1100.522,329.133,415.735,179.172,17.877,152.000
C05399=1100.530,329.512,415.686,179.177,17.880,152.000
C05400=1100.539,329.889,415.637,179.183,17.884,152.000
C05401=1100.548,330.268,415.586,179.187,17.889,152.000
C05402=1100.557,330.646,415.537,179.192,17.892,152.000
C05403=1100.562,330.894,415.504,179.196,17.895,152.000
C05404=1100.568,331.142,415.471,179.199,17.898,152.000
C05405=1100.574,331.389,415.439,179.202,17.900,152.000
C05406=1100.580,331.637,415.406,179.205,17.903,152.000
C05407=1100.586,331.885,415.374,179.208,17.906,152.000
C05408=1100.591,332.133,415.340,179.212,17.909,152.000
C05409=1100.598,332.381,415.308,179.215,17.911,152.000
C05410=1100.603,332.629,415.274,179.218,17.914,152.000
C05411=1100.608,332.876,415.243,179.221,17.917,152.000
C05412=1100.614,333.124,415.209,179.224,17.919,152.000
C05413=1100.620,333.372,415.177,179.228,17.923,152.000
C05414=1100.626,333.620,415.143,179.231,17.925,152.000
C05415=1100.631,333.868,415.111,179.234,17.928,152.000
C05416=1100.637,334.115,415.078,179.237,17.930,152.000
C05417=1100.642,334.363,415.045,179.241,17.934,152.000
C05418=1100.648,334.611,415.012,179.244,17.937,152.000
C05419=1100.654,334.858,414.979,179.247,17.939,152.000
C05420=1100.660,335.106,414.945,179.250,17.942,152.001
C05421=1100.665,335.355,414.913,179.254,17.945,152.001
C05422=1100.671,335.602,414.880,179.257,17.948,152.001
C05423=1100.676,335.850,414.847,179.260,17.950,152.001
C05424=1100.682,336.097,414.814,179.263,17.953,152.001
C05425=1100.688,336.345,414.781,179.267,17.956,152.001
C05426=1100.694,336.593,414.748,179.269,17.959,152.001
C05427=1100.699,336.841,414.714,179.272,17.962,152.001
C05428=1100.705,337.088,414.682,179.275,17.965,152.001
C05429=1100.711,337.336,414.648,179.279,17.968,152.001
C05430=1100.717,337.584,414.615,179.282,17.971,152.001
C05431=1100.723,337.832,414.582,179.285,17.974,152.001
C05432=1100.728,338.080,414.549,179.289,17.977,152.002
C05433=1100.734,338.328,414.516,179.292,17.979,152.001
C05434=1100.739,338.575,414.483,179.295,17.982,152.002
C05435=1100.745,338.822,414.449,179.298,17.985,152.002
C05436=1100.751,339.070,414.416,179.301,17.988,152.002
C05437=1100.757,339.318,414.382,179.304,17.991,152.002
C05438=1100.762,339.566,414.349,179.307,17.994,152.002
C05439=1100.768,339.813,414.316,179.311,17.998,152.002
C05440=1100.773,340.061,414.282,179.314,18.000,152.002
C05441=1100.779,340.309,414.249,179.317,18.003,152.002
C05442=1100.785,340.557,414.215,179.321,18.007,152.003
C05443=1100.790,340.804,414.182,179.323,18.010,152.003
C05444=1100.797,341.052,414.149,179.326,18.012,152.003
C05445=1100.802,341.300,414.116,179.330,18.016,152.003
C05446=1100.808,341.547,414.082,179.333,18.019,152.003
C05447=1100.814,341.795,414.048,179.336,18.021,152.003
C05448=1100.819,342.043,414.015,179.340,18.025,152.003
C05449=1100.825,342.291,413.982,179.342,18.028,152.003
